C01819=1049.638,44.373,421.280,170.592,33.562,156.310
C01820=1049.643,44.623,421.263,170.594,33.564,156.311
C01821=1049.650,44.872,421.246,170.596,33.566,156.311
C01822=1049.656,45.158,421.226,170.597,33.568,156.311
C01823=1049.664,45.444,421.207,170.599,33.571,156.312
C01824=1049.671,45.731,421.188,170.601,33.573,156.312
C01825=1049.678,46.017,421.168,170.603,33.575,156.312
C01826=1049.684,46.266,421.152,170.605,33.577,156.313
C01827=1049.690,46.516,421.134,170.606,33.579,156.313
C01828=1049.696,46.765,421.117,170.608,33.581,156.313
C01829=1049.702,47.014,421.100,170.610,33.583,156.314
C01830=1049.709,47.263,421.083,170.611,33.585,156.314
C01831=1049.714,47.513,421.066,170.613,33.587,156.314
C01832=1049.721,47.762,421.049,170.615,33.589,156.315
C01833=1049.727,48.012,421.033,170.617,33.590,156.315
C01834=1049.732,48.261,421.015,170.619,33.592,156.315
C01835=1049.739,48.510,420.998,170.620,33.594,156.316
C01836=1049.745,48.759,420.982,170.622,33.596,156.316
C01837=1049.751,49.008,420.964,170.624,33.598,156.316
C01838=1049.757,49.258,420.947,170.625,33.600,156.316
C01839=1049.763,49.507,420.930,170.627,33.602,156.317
C01840=1049.770,49.757,420.912,170.629,33.604,156.317
C01841=1049.775,50.006,420.896,170.630,33.606,156.317
C01842=1049.781,50.255,420.879,170.632,33.608,156.318
C01843=1049.788,50.505,420.861,170.634,33.610,156.318
C01844=1049.794,50.754,420.845,170.635,33.612,156.318
C01845=1049.800,51.004,420.827,170.637,33.614,156.319
C01846=1049.806,51.253,420.810,170.638,33.616,156.319
C01847=1049.813,51.503,420.793,170.640,33.618,156.319
C01848=1049.818,51.752,420.776,170.642,33.620,156.320
C01849=1049.825,52.001,420.759,170.643,33.622,156.320
C01850=1049.831,52.250,420.742,170.645,33.624,156.320
C01851=1049.837,52.499,420.725,170.647,33.626,156.321
C01852=1049.843,52.749,420.707,170.648,33.628,156.321
C01853=1049.850,52.998,420.690,170.650,33.630,156.321
C01854=1049.856,53.247,420.673,170.652,33.632,156.322
C01855=1049.862,53.497,420.656,170.653,33.633,156.322
C01856=1049.868,53.746,420.638,170.655,33.635,156.322
C01857=1049.874,53.995,420.621,170.656,33.637,156.322
C01858=1049.881,54.245,420.604,170.658,33.639,156.323
C01859=1049.886,54.494,420.587,170.660,33.641,156.323
C01860=1049.893,54.744,420.570,170.661,33.643,156.323
C01861=1049.899,54.992,420.553,170.663,33.645,156.324
C01862=1049.905,55.242,420.535,170.665,33.647,156.324
C01863=1049.912,55.491,420.518,170.666,33.649,156.324
C01864=1049.918,55.741,420.501,170.668,33.651,156.325
C01865=1049.924,55.990,420.484,170.670,33.653,156.325
C01866=1049.931,56.239,420.466,170.671,33.655,156.325
C01867=1049.936,56.488,420.449,170.673,33.657,156.326
C01868=1049.943,56.738,420.432,170.674,33.659,156.326
C01869=1049.949,56.988,420.414,170.676,33.660,156.326
C01870=1049.955,57.236,420.397,170.678,33.662,156.326
C01871=1049.962,57.486,420.380,170.679,33.664,156.327
C01872=1049.967,57.735,420.362,170.681,33.666,156.327
C01873=1049.974,57.985,420.345,170.684,33.668,156.327
C01874=1049.980,58.234,420.328,170.685,33.670,156.328
C01875=1049.987,58.483,420.310,170.687,33.672,156.328
C01876=1049.994,58.733,420.293,170.689,33.674,156.328
C01877=1049.999,58.982,420.275,170.690,33.676,156.329
C01878=1050.006,59.231,420.258,170.692,33.678,156.329
C01879=1050.011,59.480,420.240,170.693,33.680,156.329
C01880=1050.018,59.730,420.223,170.695,33.682,156.330
C01881=1050.024,59.979,420.205,170.697,33.683,156.330
C01882=1050.031,60.228,420.188,170.698,33.685,156.330
C01883=1050.038,60.478,420.171,170.700,33.687,156.330
C01884=1050.043,60.727,420.153,170.702,33.689,156.331
C01885=1050.050,60.976,420.136,170.703,33.691,156.331
C01886=1050.057,61.262,420.116,170.705,33.693,156.331
C01887=1050.064,61.548,420.096,170.707,33.696,156.332
C01888=1050.071,61.834,420.076,170.709,33.698,156.332
C01889=1050.079,62.120,420.057,170.711,33.700,156.332
C01890=1050.085,62.369,420.039,170.712,33.702,156.333
C01891=1050.091,62.619,420.021,170.714,33.704,156.333
C01892=1050.097,62.868,420.004,170.716,33.706,156.333
C01893=1050.104,63.117,419.986,170.717,33.708,156.334
C01894=1050.110,63.366,419.968,170.719,33.710,156.334
C01895=1050.117,63.615,419.951,170.721,33.712,156.334
C01896=1050.123,63.865,419.933,170.722,33.713,156.335
C01897=1050.130,64.114,419.916,170.724,33.715,156.335
C01898=1050.135,64.363,419.898,170.726,33.717,156.335
C01899=1050.142,64.613,419.881,170.727,33.719,156.336
C01900=1050.148,64.862,419.863,170.729,33.721,156.336
C01901=1050.154,65.111,419.845,170.730,33.723,156.336
C01902=1050.160,65.361,419.827,170.732,33.725,156.337
C01903=1050.167,65.610,419.809,170.734,33.727,156.337
C01904=1050.172,65.859,419.792,170.735,33.729,156.337
C01905=1050.178,66.109,419.774,170.737,33.731,156.337
C01906=1050.185,66.358,419.756,170.739,33.733,156.338
C01907=1050.191,66.607,419.739,170.741,33.734,156.338
C01908=1050.197,66.856,419.720,170.743,33.736,156.338
C01909=1050.204,67.106,419.703,170.744,33.738,156.339
C01910=1050.210,67.355,419.685,170.746,33.741,156.339
C01911=1050.216,67.605,419.667,170.748,33.743,156.340
C01912=1050.222,67.854,419.649,170.749,33.745,156.340
C01913=1050.228,68.102,419.632,170.751,33.747,156.340
C01914=1050.235,68.352,419.614,170.753,33.749,156.340
C01915=1050.241,68.602,419.596,170.754,33.751,156.341
C01916=1050.247,68.850,419.578,170.756,33.753,156.341
C01917=1050.253,69.100,419.560,170.757,33.755,156.341
C01918=1050.259,69.350,419.542,170.759,33.757,156.342
C01919=1050.265,69.599,419.525,170.761,33.759,156.342
C01920=1050.271,69.848,419.506,170.762,33.761,156.342
C01921=1050.278,70.097,419.488,170.764,33.763,156.343
C01922=1050.283,70.346,419.471,170.766,33.764,156.343
C01923=1050.290,70.596,419.452,170.767,33.766,156.343
C01924=1050.296,70.845,419.435,170.769,33.768,156.344
C01925=1050.302,71.094,419.417,170.770,33.770,156.344
C01926=1050.308,71.343,419.398,170.772,33.772,156.344
C01927=1050.314,71.593,419.380,170.774,33.774,156.345
C01928=1050.321,71.843,419.362,170.775,33.776,156.345
C01929=1050.326,72.091,419.344,170.777,33.778,156.345
C01930=1050.332,72.341,419.326,170.779,33.780,156.346
C01931=1050.339,72.590,419.308,170.780,33.783,156.346
C01932=1050.345,72.840,419.290,170.782,33.785,156.346
C01933=1050.351,73.088,419.273,170.783,33.787,156.347
C01934=1050.358,73.338,419.254,170.786,33.789,156.347
C01935=1050.364,73.587,419.236,170.788,33.791,156.347
C01936=1050.370,73.836,419.218,170.789,33.792,156.348
C01937=1050.376,74.085,419.200,170.791,33.794,156.348
C01938=1050.382,74.335,419.181,170.792,33.796,156.348
C01939=1050.388,74.584,419.163,170.794,33.798,156.349
C01940=1050.395,74.833,419.145,170.796,33.800,156.349
C01941=1050.400,75.082,419.127,170.797,33.802,156.349
C01942=1050.407,75.332,419.108,170.799,33.804,156.350
C01943=1050.413,75.581,419.091,170.801,33.806,156.350
C01944=1050.419,75.830,419.072,170.802,33.808,156.350
C01945=1050.425,76.079,419.054,170.804,33.810,156.351
C01946=1050.431,76.329,419.036,170.805,33.812,156.351
C01947=1050.437,76.578,419.018,170.807,33.814,156.351
C01948=1050.444,76.827,419.000,170.809,33.816,156.352
C01949=1050.451,77.077,418.982,170.810,33.819,156.352
C01950=1050.457,77.363,418.960,170.812,33.821,156.352
C01951=1050.464,77.648,418.940,170.814,33.823,156.353
C01952=1050.471,77.933,418.919,170.816,33.825,156.353
C01953=1050.479,78.219,418.898,170.818,33.828,156.353
C01954=1050.484,78.468,418.880,170.819,33.830,156.354
C01955=1050.491,78.718,418.861,170.821,33.832,156.354
C01956=1050.496,78.967,418.842,170.823,33.834,156.354
C01957=1050.503,79.217,418.824,170.824,33.835,156.355
C01958=1050.509,79.466,418.805,170.827,33.837,156.355
C01959=1050.515,79.714,418.787,170.828,33.839,156.355
C01960=1050.521,79.964,418.769,170.830,33.842,156.356
C01961=1050.527,80.213,418.751,170.832,33.844,156.356
C01962=1050.533,80.463,418.731,170.833,33.846,156.357
C01963=1050.539,80.712,418.713,170.835,33.848,156.357
C01964=1050.545,80.961,418.695,170.837,33.850,156.357
C01965=1050.551,81.210,418.677,170.838,33.852,156.357
C01966=1050.558,81.460,418.659,170.840,33.854,156.358
C01967=1050.563,81.709,418.639,170.841,33.856,156.358
C01968=1050.570,81.958,418.621,170.843,33.858,156.359
C01969=1050.576,82.207,418.602,170.845,33.860,156.359
C01970=1050.582,82.456,418.584,170.846,33.862,156.359
C01971=1050.588,82.705,418.566,170.848,33.864,156.360
C01972=1050.594,82.955,418.547,170.849,33.866,156.360
C01973=1050.600,83.204,418.528,170.851,33.868,156.360
C01974=1050.606,83.454,418.510,170.853,33.871,156.361
C01975=1050.613,83.703,418.491,170.854,33.872,156.361
C01976=1050.618,83.952,418.472,170.856,33.874,156.361
C01977=1050.624,84.201,418.454,170.858,33.876,156.362
C01978=1050.630,84.450,418.436,170.859,33.878,156.362
C01979=1050.637,84.700,418.417,170.861,33.880,156.362
C01980=1050.643,84.949,418.399,170.863,33.882,156.363
C01981=1050.649,85.198,418.379,170.865,33.884,156.363
C01982=1050.655,85.447,418.361,170.867,33.887,156.363
C01983=1050.662,85.696,418.342,170.868,33.889,156.364
C01984=1050.668,85.946,418.324,170.870,33.891,156.364
C01985=1050.674,86.196,418.305,170.872,33.893,156.364
C01986=1050.680,86.445,418.286,170.873,33.895,156.365
C01987=1050.686,86.693,418.268,170.875,33.896,156.365
C01988=1050.692,86.942,418.249,170.876,33.898,156.365
C01989=1050.699,87.191,418.231,170.878,33.900,156.366
C01990=1050.704,87.441,418.211,170.880,33.902,156.366
C01991=1050.711,87.690,418.193,170.881,33.905,156.366
C01992=1050.717,87.940,418.175,170.883,33.907,156.367
C01993=1050.723,88.189,418.156,170.885,33.909,156.367
C01994=1050.729,88.438,418.137,170.886,33.911,156.367
C01995=1050.735,88.687,418.118,170.888,33.913,156.368
C01996=1050.742,88.936,418.100,170.890,33.915,156.368
C01997=1050.748,89.186,418.081,170.891,33.917,156.368
C01998=1050.754,89.435,418.062,170.893,33.919,156.369
C01999=1050.760,89.684,418.043,170.894,33.920,156.369
C02000=1050.767,89.933,418.024,170.896,33.922,156.369
C02001=1050.772,90.183,418.005,170.898,33.924,156.370
C02002=1050.779,90.432,417.987,170.900,33.926,156.370
C02003=1050.785,90.681,417.968,170.902,33.929,156.370
C02004=1050.791,90.930,417.949,170.904,33.931,156.371
C02005=1050.797,91.179,417.930,170.905,33.933,156.371
C02006=1050.803,91.429,417.911,170.907,33.935,156.371
C02007=1050.810,91.678,417.892,170.908,33.937,156.372
C02008=1050.815,91.927,417.873,170.910,33.939,156.372
C02009=1050.822,92.177,417.854,170.912,33.941,156.372
C02010=1050.827,92.426,417.835,170.913,33.943,156.373
C02011=1050.834,92.675,417.816,170.915,33.945,156.373
C02012=1050.840,92.924,417.796,170.917,33.948,156.374
C02013=1050.846,93.173,417.778,170.918,33.950,156.374
C02014=1050.853,93.459,417.756,170.920,33.952,156.374
C02015=1050.860,93.744,417.734,170.922,33.954,156.375
C02016=1050.867,94.030,417.713,170.924,33.957,156.375
C02017=1050.874,94.315,417.691,170.926,33.959,156.375
C02018=1050.879,94.564,417.672,170.927,33.961,156.376
C02019=1050.886,94.814,417.653,170.929,33.963,156.376
C02020=1050.891,95.063,417.634,170.932,33.965,156.376
C02021=1050.897,95.312,417.614,170.933,33.967,156.377
C02022=1050.904,95.562,417.595,170.935,33.969,156.377
C02023=1050.910,95.811,417.576,170.937,33.972,156.378
C02024=1050.916,96.060,417.557,170.938,33.973,156.378
C02025=1050.922,96.310,417.538,170.940,33.975,156.378
C02026=1050.929,96.558,417.518,170.941,33.977,156.379
C02027=1050.935,96.808,417.499,170.943,33.979,156.379
C02028=1050.941,97.057,417.480,170.945,33.981,156.379
C02029=1050.947,97.306,417.461,170.946,33.984,156.380
C02030=1050.953,97.555,417.442,170.948,33.986,156.380
C02031=1050.959,97.804,417.423,170.950,33.988,156.380
C02032=1050.965,98.053,417.403,170.951,33.990,156.381
C02033=1050.971,98.303,417.385,170.953,33.992,156.381
C02034=1050.977,98.552,417.365,170.955,33.994,156.381
C02035=1050.984,98.801,417.346,170.956,33.996,156.382
C02036=1050.989,99.050,417.327,170.958,33.998,156.382
C02037=1050.996,99.300,417.308,170.960,34.000,156.382
C02038=1051.002,99.549,417.288,170.962,34.002,156.383
C02039=1051.009,99.798,417.269,170.964,34.004,156.383
C02040=1051.014,100.047,417.250,170.966,34.006,156.383
C02041=1051.020,100.296,417.230,170.967,34.008,156.384
C02042=1051.027,100.545,417.211,170.969,34.010,156.384
C02043=1051.033,100.795,417.192,170.970,34.012,156.384
C02044=1051.039,101.043,417.172,170.972,34.014,156.385
C02045=1051.045,101.292,417.153,170.974,34.016,156.385
C02046=1051.051,101.542,417.134,170.975,34.019,156.386
C02047=1051.057,101.791,417.114,170.977,34.021,156.386
C02048=1051.063,102.041,417.095,170.979,34.023,156.386
C02049=1051.069,102.290,417.075,170.980,34.024,156.387
C02050=1051.075,102.539,417.056,170.982,34.027,156.387
C02051=1051.081,102.788,417.036,170.984,34.029,156.387
C02052=1051.087,103.037,417.017,170.985,34.031,156.388
C02053=1051.093,103.286,416.997,170.987,34.033,156.388
C02054=1051.099,103.535,416.978,170.989,34.035,156.388
C02055=1051.105,103.784,416.958,170.991,34.037,156.389
C02056=1051.111,104.033,416.939,170.993,34.039,156.389
C02057=1051.117,104.283,416.919,170.995,34.042,156.389
C02058=1051.123,104.532,416.899,170.996,34.044,156.390
C02059=1051.129,104.782,416.880,170.998,34.046,156.390
C02060=1051.135,105.030,416.860,170.999,34.048,156.390
C02061=1051.142,105.279,416.841,171.001,34.050,156.391
C02062=1051.148,105.528,416.822,171.003,34.052,156.391
C02063=1051.154,105.777,416.802,171.004,34.054,156.392
C02064=1051.160,106.027,416.782,171.006,34.056,156.392
C02065=1051.166,106.276,416.762,171.008,34.059,156.392
C02066=1051.172,106.526,416.743,171.009,34.060,156.393
C02067=1051.178,106.774,416.724,171.011,34.062,156.393
C02068=1051.184,107.023,416.704,171.013,34.064,156.393
C02069=1051.191,107.273,416.684,171.014,34.066,156.394
C02070=1051.197,107.522,416.664,171.016,34.069,156.394
C02071=1051.202,107.771,416.645,171.019,34.071,156.394
C02072=1051.208,108.020,416.625,171.020,34.073,156.395
C02073=1051.215,108.269,416.606,171.022,34.075,156.395
C02074=1051.221,108.519,416.586,171.024,34.077,156.396
C02075=1051.227,108.767,416.566,171.025,34.079,156.396
C02076=1051.233,109.017,416.547,171.027,34.081,156.396
C02077=1051.239,109.266,416.527,171.029,34.083,156.397
C02078=1051.246,109.551,416.504,171.031,34.086,156.397
C02079=1051.253,109.837,416.481,171.033,34.088,156.397
C02080=1051.260,110.123,416.459,171.035,34.090,156.398
C02081=1051.267,110.408,416.436,171.036,34.093,156.398
C02082=1051.274,110.658,416.417,171.038,34.095,156.399
C02083=1051.280,110.906,416.397,171.040,34.097,156.399
C02084=1051.286,111.155,416.377,171.041,34.099,156.399
C02085=1051.292,111.405,416.358,171.043,34.101,156.400
C02086=1051.298,111.654,416.337,171.045,34.103,156.400
C02087=1051.304,111.903,416.317,171.048,34.105,156.400
C02088=1051.310,112.152,416.297,171.049,34.107,156.401
C02089=1051.316,112.401,416.278,171.051,34.109,156.401
C02090=1051.322,112.651,416.258,171.053,34.111,156.401
C02091=1051.328,112.900,416.238,171.054,34.114,156.402
C02092=1051.334,113.148,416.218,171.056,34.116,156.402
C02093=1051.340,113.397,416.198,171.058,34.118,156.402
C02094=1051.347,113.647,416.178,171.059,34.120,156.403
C02095=1051.353,113.896,416.158,171.061,34.122,156.403
C02096=1051.358,114.145,416.138,171.063,34.124,156.404
C02097=1051.364,114.394,416.118,171.064,34.126,156.404
C02098=1051.371,114.644,416.097,171.066,34.129,156.404
C02099=1051.377,114.892,416.078,171.068,34.131,156.405
C02100=1051.382,115.142,416.057,171.069,34.133,156.405
C02101=1051.388,115.390,416.037,171.072,34.135,156.405
C02102=1051.394,115.641,416.017,171.074,34.137,156.406
C02103=1051.399,115.890,415.997,171.075,34.139,156.406
C02104=1051.405,116.138,415.977,171.077,34.141,156.407
C02105=1051.411,116.387,415.957,171.079,34.144,156.407
C02106=1051.418,116.637,415.937,171.080,34.146,156.407
C02107=1051.423,116.886,415.916,171.082,34.148,156.408
C02108=1051.429,117.135,415.896,171.084,34.150,156.408
C02109=1051.436,117.384,415.876,171.085,34.152,156.408
C02110=1051.442,117.633,415.856,171.087,34.154,156.409
C02111=1051.447,117.882,415.835,171.089,34.157,156.409
C02112=1051.453,118.131,415.815,171.090,34.159,156.410
C02113=1051.460,118.381,415.795,171.092,34.161,156.410
C02114=1051.466,118.629,415.775,171.094,34.163,156.410
C02115=1051.471,118.878,415.754,171.096,34.165,156.411
C02116=1051.477,119.128,415.734,171.098,34.168,156.411
C02117=1051.483,119.377,415.714,171.100,34.170,156.411
C02118=1051.489,119.626,415.694,171.102,34.172,156.412
C02119=1051.495,119.875,415.673,171.103,34.174,156.412
C02120=1051.501,120.124,415.653,171.105,34.176,156.413
C02121=1051.507,120.373,415.633,171.107,34.179,156.413
C02122=1051.513,120.623,415.612,171.108,34.180,156.413
C02123=1051.519,120.871,415.592,171.110,34.182,156.414
C02124=1051.525,121.120,415.572,171.112,34.185,156.414
C02125=1051.531,121.370,415.551,171.113,34.187,156.414
C02126=1051.537,121.619,415.531,171.115,34.189,156.415
C02127=1051.543,121.867,415.511,171.117,34.191,156.415
C02128=1051.549,122.117,415.490,171.119,34.193,156.416
C02129=1051.555,122.366,415.470,171.121,34.195,156.416
C02130=1051.562,122.615,415.450,171.123,34.198,156.416
C02131=1051.567,122.864,415.429,171.125,34.200,156.417
C02132=1051.573,123.113,415.409,171.126,34.202,156.417
C02133=1051.580,123.362,415.388,171.128,34.204,156.417
C02134=1051.585,123.611,415.368,171.130,34.206,156.418
C02135=1051.592,123.861,415.347,171.132,34.208,156.418
C02136=1051.598,124.110,415.327,171.133,34.211,156.419
C02137=1051.604,124.358,415.307,171.135,34.212,156.419
C02138=1051.610,124.608,415.286,171.137,34.214,156.419
C02139=1051.616,124.857,415.266,171.138,34.217,156.420
C02140=1051.622,125.106,415.246,171.140,34.219,156.420
C02141=1051.628,125.355,415.225,171.142,34.221,156.420
C02142=1051.635,125.641,415.201,171.145,34.223,156.421
C02143=1051.642,125.926,415.178,171.147,34.226,156.421
C02144=1051.649,126.211,415.154,171.149,34.228,156.422
C02145=1051.656,126.497,415.130,171.151,34.231,156.422
C02146=1051.662,126.746,415.110,171.153,34.233,156.422
C02147=1051.668,126.995,415.090,171.154,34.235,156.423
C02148=1051.675,127.244,415.068,171.156,34.237,156.423
C02149=1051.681,127.493,415.048,171.158,34.239,156.423
C02150=1051.687,127.743,415.028,171.160,34.241,156.424
C02151=1051.693,127.991,415.007,171.161,34.243,156.424
C02152=1051.699,128.241,414.987,171.163,34.246,156.425
C02153=1051.705,128.490,414.966,171.165,34.248,156.425
C02154=1051.711,128.739,414.945,171.167,34.250,156.425
C02155=1051.717,128.988,414.925,171.169,34.252,156.426
C02156=1051.723,129.237,414.904,171.171,34.254,156.426
C02157=1051.730,129.486,414.883,171.173,34.256,156.426
C02158=1051.736,129.735,414.863,171.175,34.259,156.427
C02159=1051.741,129.984,414.843,171.176,34.260,156.427
C02160=1051.748,130.233,414.821,171.178,34.262,156.427
C02161=1051.754,130.482,414.802,171.180,34.265,156.428
C02162=1051.760,130.731,414.780,171.182,34.267,156.428
C02163=1051.766,130.980,414.760,171.183,34.269,156.429
C02164=1051.772,131.230,414.739,171.185,34.271,156.429
C02165=1051.779,131.479,414.718,171.187,34.273,156.429
C02166=1051.784,131.728,414.697,171.189,34.275,156.430
C02167=1051.791,131.977,414.676,171.191,34.278,156.430
C02168=1051.797,132.226,414.656,171.193,34.280,156.430
C02169=1051.803,132.475,414.634,171.195,34.282,156.431
C02170=1051.809,132.724,414.614,171.197,34.284,156.431
C02171=1051.815,132.973,414.593,171.198,34.286,156.432
C02172=1051.820,133.222,414.572,171.200,34.289,156.432
C02173=1051.827,133.471,414.551,171.202,34.290,156.432
C02174=1051.833,133.720,414.530,171.204,34.293,156.433
C02175=1051.839,133.969,414.509,171.205,34.295,156.433
C02176=1051.845,134.218,414.488,171.207,34.297,156.434
C02177=1051.851,134.467,414.467,171.209,34.299,156.434
C02178=1051.857,134.717,414.446,171.211,34.301,156.434
C02179=1051.863,134.965,414.426,171.213,34.304,156.435
C02180=1051.869,135.215,414.404,171.215,34.306,156.435
C02181=1051.875,135.463,414.383,171.217,34.308,156.436
C02182=1051.881,135.713,414.362,171.219,34.310,156.436
C02183=1051.887,135.961,414.341,171.221,34.313,156.436
C02184=1051.893,136.210,414.319,171.222,34.315,156.437
C02185=1051.900,136.460,414.299,171.224,34.317,156.437
C02186=1051.905,136.708,414.278,171.226,34.319,156.437
C02187=1051.911,136.958,414.256,171.228,34.321,156.438
C02188=1051.917,137.206,414.236,171.229,34.324,156.438
C02189=1051.923,137.456,414.215,171.231,34.325,156.439
C02190=1051.930,137.705,414.193,171.233,34.328,156.439
C02191=1051.935,137.954,414.172,171.236,34.330,156.439
C02192=1051.942,138.203,414.151,171.238,34.332,156.440
C02193=1051.947,138.451,414.130,171.239,34.334,156.440
C02194=1051.953,138.700,414.109,171.241,34.336,156.440
C02195=1051.959,138.950,414.088,171.243,34.339,156.441
C02196=1051.966,139.199,414.067,171.245,34.341,156.441
C02197=1051.972,139.448,414.045,171.246,34.343,156.442
C02198=1051.978,139.697,414.024,171.248,34.345,156.442
C02199=1051.983,139.946,414.003,171.250,34.348,156.442
C02200=1051.989,140.195,413.981,171.252,34.350,156.443
C02201=1051.995,140.444,413.960,171.254,34.352,156.443
C02202=1052.001,140.693,413.939,171.256,34.354,156.444
C02203=1052.008,140.942,413.918,171.258,34.357,156.444
C02204=1052.013,141.191,413.897,171.260,34.359,156.444
C02205=1052.019,141.440,413.875,171.262,34.361,156.445
C02206=1052.026,141.725,413.850,171.264,34.364,156.445
C02207=1052.033,142.010,413.826,171.266,34.366,156.446
C02208=1052.040,142.296,413.802,171.268,34.369,156.446
C02209=1052.047,142.582,413.776,171.270,34.371,156.447
C02210=1052.052,142.830,413.755,171.272,34.373,156.447
C02211=1052.059,143.079,413.734,171.274,34.376,156.447
C02212=1052.065,143.329,413.713,171.276,34.378,156.448
C02213=1052.071,143.577,413.692,171.278,34.380,156.448
C02214=1052.077,143.826,413.670,171.280,34.382,156.448
C02215=1052.083,144.076,413.649,171.282,34.385,156.449
C02216=1052.088,144.324,413.627,171.284,34.387,156.449
C02217=1052.095,144.573,413.606,171.285,34.389,156.450
C02218=1052.101,144.823,413.584,171.287,34.392,156.450
C02219=1052.106,145.071,413.563,171.289,34.393,156.450
C02220=1052.113,145.320,413.541,171.291,34.396,156.451
C02221=1052.119,145.569,413.520,171.293,34.398,156.451
C02222=1052.125,145.819,413.498,171.295,34.400,156.452
C02223=1052.130,146.067,413.477,171.297,34.402,156.452
C02224=1052.137,146.316,413.455,171.299,34.405,156.453
C02225=1052.143,146.566,413.433,171.301,34.407,156.453
C02226=1052.149,146.815,413.412,171.303,34.409,156.453
C02227=1052.154,147.063,413.390,171.305,34.411,156.454
C02228=1052.161,147.313,413.369,171.307,34.414,156.454
C02229=1052.167,147.562,413.347,171.308,34.416,156.454
C02230=1052.173,147.810,413.325,171.310,34.418,156.455
C02231=1052.179,148.059,413.304,171.312,34.420,156.455
C02232=1052.185,148.308,413.282,171.314,34.423,156.456
C02233=1052.191,148.557,413.260,171.317,34.425,156.456
C02234=1052.197,148.806,413.239,171.319,34.427,156.456
C02235=1052.203,149.055,413.217,171.320,34.430,156.457
C02236=1052.209,149.304,413.196,171.322,34.432,156.457
C02237=1052.215,149.553,413.173,171.324,34.434,156.458
C02238=1052.221,149.802,413.151,171.326,34.436,156.458
C02239=1052.226,150.051,413.130,171.328,34.439,156.458
C02240=1052.233,150.300,413.108,171.330,34.440,156.459
C02241=1052.239,150.549,413.087,171.332,34.443,156.459
C02242=1052.245,150.798,413.064,171.333,34.445,156.460
C02243=1052.251,151.047,413.042,171.336,34.447,156.460
C02244=1052.256,151.296,413.021,171.338,34.450,156.460
C02245=1052.262,151.545,412.999,171.340,34.452,156.461
C02246=1052.269,151.794,412.978,171.342,34.454,156.461
C02247=1052.275,152.043,412.955,171.344,34.457,156.462
C02248=1052.280,152.292,412.933,171.345,34.459,156.462
C02249=1052.286,152.541,412.912,171.347,34.461,156.463
C02250=1052.293,152.789,412.889,171.349,34.463,156.463
C02251=1052.299,153.039,412.868,171.351,34.466,156.463
C02252=1052.305,153.288,412.846,171.353,34.468,156.464
C02253=1052.311,153.537,412.823,171.356,34.470,156.464
C02254=1052.317,153.786,412.801,171.358,34.473,156.465
C02255=1052.322,154.034,412.780,171.360,34.475,156.465
C02256=1052.329,154.283,412.758,171.361,34.477,156.465
C02257=1052.335,154.532,412.736,171.363,34.480,156.466
C02258=1052.340,154.782,412.714,171.365,34.482,156.466
C02259=1052.347,155.030,412.692,171.367,34.484,156.467
C02260=1052.353,155.279,412.670,171.369,34.487,156.467
C02261=1052.358,155.529,412.648,171.371,34.489,156.467
C02262=1052.364,155.777,412.626,171.373,34.491,156.468
C02263=1052.370,156.026,412.604,171.376,34.494,156.468
C02264=1052.376,156.275,412.581,171.377,34.495,156.469
C02265=1052.382,156.524,412.560,171.379,34.498,156.469
C02266=1052.389,156.773,412.537,171.381,34.501,156.470
C02267=1052.394,157.022,412.515,171.383,34.502,156.470
C02268=1052.401,157.271,412.493,171.385,34.505,156.470
C02269=1052.406,157.520,412.470,171.387,34.507,156.471
C02270=1052.413,157.805,412.445,171.389,34.510,156.471
C02271=1052.420,158.090,412.420,171.391,34.513,156.472
C02272=1052.426,158.375,412.395,171.394,34.515,156.472
C02273=1052.434,158.660,412.369,171.397,34.518,156.473
C02274=1052.440,158.909,412.347,171.399,34.520,156.473
C02275=1052.446,159.158,412.325,171.400,34.523,156.473
C02276=1052.451,159.407,412.303,171.402,34.525,156.474
C02277=1052.458,159.655,412.281,171.404,34.527,156.474
C02278=1052.463,159.904,412.258,171.406,34.530,156.475
C02279=1052.469,160.153,412.236,171.408,34.531,156.475
C02280=1052.476,160.402,412.214,171.411,34.534,156.475
C02281=1052.481,160.652,412.191,171.413,34.537,156.476
C02282=1052.488,160.900,412.169,171.415,34.538,156.476
C02283=1052.494,161.149,412.146,171.417,34.541,156.477
C02284=1052.499,161.399,412.124,171.419,34.543,156.477
C02285=1052.505,161.647,412.101,171.421,34.546,156.478
C02286=1052.511,161.896,412.079,171.422,34.548,156.478
C02287=1052.517,162.146,412.056,171.424,34.551,156.479
C02288=1052.522,162.394,412.033,171.426,34.554,156.479
C02289=1052.527,162.643,412.011,171.429,34.555,156.479
C02290=1052.534,162.891,411.988,171.431,34.558,156.480
C02291=1052.539,163.141,411.966,171.433,34.560,156.480
C02292=1052.545,163.390,411.943,171.435,34.563,156.481
C02293=1052.551,163.639,411.920,171.437,34.565,156.481
C02294=1052.557,163.887,411.898,171.439,34.568,156.482
C02295=1052.563,164.137,411.876,171.441,34.571,156.482
C02296=1052.568,164.386,411.853,171.442,34.573,156.483
C02297=1052.574,164.634,411.830,171.445,34.575,156.483
C02298=1052.581,164.883,411.808,171.447,34.577,156.483
C02299=1052.586,165.132,411.785,171.449,34.580,156.484
C02300=1052.592,165.381,411.762,171.451,34.582,156.484
C02301=1052.598,165.630,411.739,171.453,34.585,156.485
C02302=1052.603,165.879,411.716,171.455,34.587,156.485
C02303=1052.610,166.128,411.694,171.457,34.590,156.486
C02304=1052.615,166.377,411.671,171.459,34.592,156.486
C02305=1052.621,166.626,411.648,171.461,34.594,156.486
C02306=1052.627,166.875,411.625,171.464,34.597,156.487
C02307=1052.633,167.123,411.603,171.466,34.599,156.487
C02308=1052.639,167.372,411.580,171.468,34.602,156.488
C02309=1052.645,167.622,411.558,171.470,34.604,156.488
C02310=1052.650,167.870,411.535,171.472,34.607,156.489
C02311=1052.656,168.119,411.512,171.474,34.610,156.489
C02312=1052.662,168.368,411.489,171.476,34.611,156.489
C02313=1052.668,168.617,411.467,171.477,34.614,156.490
C02314=1052.674,168.866,411.444,171.480,34.616,156.490
C02315=1052.680,169.115,411.421,171.482,34.619,156.491
C02316=1052.685,169.364,411.398,171.484,34.621,156.491
C02317=1052.691,169.612,411.375,171.486,34.624,156.492
C02318=1052.698,169.861,411.352,171.488,34.626,156.492
C02319=1052.703,170.110,411.329,171.490,34.628,156.493
C02320=1052.709,170.359,411.307,171.492,34.631,156.493
C02321=1052.715,170.608,411.284,171.494,34.633,156.493
C02322=1052.721,170.857,411.261,171.497,34.636,156.494
C02323=1052.727,171.105,411.238,171.499,34.638,156.494
C02324=1052.733,171.355,411.215,171.501,34.641,156.495
C02325=1052.739,171.603,411.191,171.503,34.643,156.495
C02326=1052.745,171.852,411.168,171.505,34.646,156.496
C02327=1052.751,172.101,411.145,171.507,34.648,156.496
C02328=1052.757,172.350,411.122,171.509,34.650,156.497
C02329=1052.763,172.598,411.100,171.511,34.653,156.497
C02330=1052.769,172.847,411.077,171.514,34.655,156.497
C02331=1052.774,173.096,411.054,171.516,34.658,156.498
C02332=1052.781,173.346,411.031,171.518,34.660,156.498
C02333=1052.787,173.595,411.008,171.520,34.663,156.499
C02334=1052.794,173.878,410.982,171.523,34.665,156.499
C02335=1052.800,174.163,410.955,171.525,34.669,156.500
C02336=1052.808,174.448,410.929,171.527,34.671,156.500
C02337=1052.814,174.732,410.902,171.530,34.674,156.501
C02338=1052.820,174.981,410.879,171.532,34.676,156.501
C02339=1052.826,175.230,410.857,171.534,34.679,156.502
C02340=1052.832,175.478,410.833,171.537,34.681,156.502
C02341=1052.838,175.728,410.810,171.539,34.684,156.503
C02342=1052.844,175.977,410.787,171.541,34.686,156.503
C02343=1052.850,176.226,410.764,171.543,34.689,156.504
C02344=1052.856,176.474,410.740,171.546,34.691,156.504
C02345=1052.862,176.724,410.717,171.548,34.694,156.504
C02346=1052.868,176.972,410.694,171.550,34.696,156.505
C02347=1052.875,177.220,410.671,171.552,34.698,156.505
C02348=1052.880,177.469,410.648,171.554,34.701,156.506
C02349=1052.887,177.719,410.625,171.556,34.703,156.506
C02350=1052.893,177.967,410.601,171.558,34.706,156.507
C02351=1052.899,178.216,410.578,171.560,34.708,156.507
C02352=1052.904,178.465,410.555,171.563,34.711,156.508
C02353=1052.911,178.714,410.531,171.565,34.713,156.508
C02354=1052.917,178.963,410.508,171.567,34.716,156.508
C02355=1052.922,179.212,410.485,171.569,34.717,156.509
C02356=1052.929,179.461,410.461,171.571,34.720,156.509
C02357=1052.936,179.709,410.439,171.573,34.722,156.510
C02358=1052.941,179.958,410.416,171.575,34.725,156.510
C02359=1052.947,180.206,410.392,171.578,34.727,156.511
C02360=1052.954,180.456,410.369,171.581,34.730,156.511
C02361=1052.960,180.704,410.345,171.583,34.732,156.512
C02362=1052.965,180.953,410.322,171.585,34.735,156.512
C02363=1052.972,181.202,410.298,171.587,34.737,156.512
C02364=1052.978,181.451,410.275,171.589,34.740,156.513
C02365=1052.984,181.699,410.252,171.591,34.742,156.513
C02366=1052.990,181.949,410.229,171.593,34.744,156.514
C02367=1052.996,182.197,410.205,171.596,34.747,156.514
C02368=1053.002,182.447,410.182,171.598,34.749,156.515
C02369=1053.009,182.695,410.158,171.600,34.752,156.515
C02370=1053.015,182.944,410.136,171.603,34.754,156.516
C02371=1053.022,183.193,410.112,171.605,34.757,156.516
C02372=1053.027,183.442,410.089,171.607,34.759,156.516
C02373=1053.033,183.690,410.065,171.609,34.762,156.517
C02374=1053.040,183.939,410.042,171.612,34.764,156.517
C02375=1053.046,184.188,410.018,171.614,34.767,156.518
C02376=1053.051,184.438,409.994,171.616,34.769,156.518
C02377=1053.057,184.686,409.970,171.618,34.772,156.519
C02378=1053.063,184.935,409.946,171.620,34.774,156.519
C02379=1053.068,185.183,409.923,171.622,34.777,156.520
C02380=1053.075,185.432,409.899,171.625,34.780,156.520
C02381=1053.080,185.681,409.875,171.628,34.783,156.521
C02382=1053.086,185.929,409.851,171.630,34.785,156.521
C02383=1053.092,186.179,409.827,171.632,34.788,156.522
C02384=1053.098,186.427,409.804,171.634,34.791,156.522
C02385=1053.103,186.676,409.779,171.636,34.793,156.523
C02386=1053.110,186.925,409.755,171.638,34.796,156.523
C02387=1053.115,187.174,409.732,171.641,34.798,156.524
C02388=1053.121,187.422,409.708,171.643,34.801,156.524
C02389=1053.127,187.672,409.684,171.645,34.804,156.525
C02390=1053.133,187.920,409.660,171.648,34.806,156.525
C02391=1053.139,188.168,409.636,171.650,34.809,156.526
C02392=1053.145,188.418,409.612,171.652,34.811,156.526
C02393=1053.151,188.667,409.589,171.654,34.814,156.527
C02394=1053.156,188.916,409.564,171.657,34.817,156.527
C02395=1053.163,189.164,409.540,171.659,34.819,156.528
C02396=1053.168,189.413,409.516,171.661,34.822,156.528
C02397=1053.174,189.662,409.492,171.663,34.825,156.529
C02398=1053.181,189.946,409.465,171.666,34.827,156.529
C02399=1053.188,190.229,409.437,171.668,34.830,156.530
C02400=1053.194,190.514,409.409,171.672,34.834,156.530
C02401=1053.201,190.798,409.382,171.674,34.837,156.531
C02402=1053.207,191.047,409.358,171.676,34.839,156.531
C02403=1053.212,191.296,409.334,171.678,34.842,156.532
C02404=1053.218,191.544,409.310,171.681,34.845,156.532
C02405=1053.224,191.794,409.286,171.683,34.847,156.533
C02406=1053.230,192.042,409.262,171.686,34.850,156.533
C02407=1053.236,192.291,409.238,171.688,34.853,156.534
C02408=1053.242,192.540,409.214,171.690,34.855,156.534
C02409=1053.248,192.789,409.189,171.692,34.858,156.535
C02410=1053.254,193.037,409.166,171.695,34.860,156.535
C02411=1053.260,193.286,409.141,171.697,34.863,156.536
C02412=1053.266,193.534,409.117,171.700,34.866,156.536
C02413=1053.272,193.783,409.092,171.702,34.868,156.537
C02414=1053.278,194.032,409.068,171.704,34.871,156.537
C02415=1053.284,194.281,409.044,171.706,34.874,156.538
C02416=1053.290,194.529,409.020,171.709,34.876,156.538
C02417=1053.296,194.779,408.995,171.711,34.879,156.539
C02418=1053.302,195.027,408.972,171.714,34.882,156.539
C02419=1053.308,195.276,408.947,171.716,34.885,156.540
C02420=1053.314,195.524,408.924,171.718,34.887,156.540
C02421=1053.320,195.774,408.899,171.721,34.890,156.541
C02422=1053.327,196.022,408.874,171.723,34.893,156.541
C02423=1053.332,196.271,408.850,171.725,34.895,156.542
C02424=1053.338,196.520,408.825,171.728,34.898,156.542
C02425=1053.344,196.768,408.802,171.730,34.901,156.543
C02426=1053.350,197.017,408.777,171.733,34.903,156.543
C02427=1053.357,197.266,408.752,171.735,34.906,156.544
C02428=1053.362,197.514,408.728,171.737,34.909,156.544
C02429=1053.369,197.763,408.704,171.739,34.911,156.545
C02430=1053.374,198.012,408.680,171.743,34.914,156.545
C02431=1053.381,198.261,408.654,171.745,34.917,156.546
C02432=1053.387,198.510,408.630,171.747,34.919,156.546
C02433=1053.393,198.758,408.606,171.749,34.922,156.547
C02434=1053.399,199.007,408.582,171.752,34.925,156.547
C02435=1053.405,199.256,408.557,171.754,34.927,156.548
C02436=1053.411,199.504,408.533,171.757,34.930,156.548
C02437=1053.417,199.753,408.508,171.759,34.933,156.549
C02438=1053.423,200.001,408.483,171.761,34.935,156.549
C02439=1053.430,200.250,408.459,171.764,34.938,156.550
C02440=1053.435,200.500,408.435,171.766,34.941,156.550
C02441=1053.442,200.748,408.410,171.768,34.943,156.551
C02442=1053.448,200.997,408.386,171.772,34.946,156.551
C02443=1053.454,201.246,408.361,171.774,34.949,156.552
C02444=1053.461,201.494,408.336,171.776,34.952,156.552
C02445=1053.466,201.743,408.312,171.778,34.954,156.553
C02446=1053.472,201.991,408.287,171.781,34.957,156.553
C02447=1053.478,202.241,408.262,171.783,34.960,156.554
C02448=1053.484,202.488,408.238,171.786,34.963,156.554
C02449=1053.490,202.738,408.213,171.788,34.965,156.555
C02450=1053.496,202.986,408.188,171.791,34.968,156.555
C02451=1053.502,203.235,408.164,171.793,34.971,156.556
C02452=1053.508,203.484,408.138,171.795,34.974,156.556
C02453=1053.514,203.733,408.114,171.798,34.977,156.557
C02454=1053.519,203.981,408.089,171.801,34.979,156.557
C02455=1053.525,204.230,408.064,171.803,34.982,156.558
C02456=1053.532,204.479,408.039,171.805,34.985,156.558
C02457=1053.538,204.727,408.014,171.807,34.988,156.559
C02458=1053.544,204.976,407.990,171.810,34.991,156.560
C02459=1053.550,205.224,407.964,171.813,34.994,156.560
C02460=1053.556,205.473,407.939,171.815,34.997,156.561
C02461=1053.561,205.722,407.915,171.818,34.999,156.561
C02462=1053.587,206.773,407.809,172.030,35.092,156.577
C02463=1053.594,207.017,407.784,172.033,35.096,156.578
C02464=1053.599,207.260,407.758,172.034,35.100,156.578
C02465=1053.606,207.504,407.733,172.036,35.103,156.579
C02466=1053.612,207.747,407.707,172.038,35.106,156.580
C02467=1053.618,207.991,407.682,172.040,35.110,156.580
C02468=1053.624,208.235,407.656,172.042,35.113,156.581
C02469=1053.630,208.478,407.632,172.044,35.117,156.582
C02470=1053.637,208.722,407.606,172.045,35.121,156.582
C02471=1053.643,208.971,407.580,172.048,35.124,156.583
C02472=1053.649,209.219,407.554,172.050,35.128,156.584
C02473=1053.656,209.467,407.527,172.052,35.132,156.585
C02474=1053.662,209.716,407.501,172.054,35.135,156.585
C02475=1053.668,209.965,407.475,172.056,35.139,156.586
C02476=1053.675,210.213,407.450,172.058,35.142,156.587
C02477=1053.681,210.462,407.423,172.059,35.146,156.587
C02478=1053.687,210.710,407.397,172.062,35.150,156.588
C02479=1053.694,210.959,407.372,172.064,35.153,156.589
C02480=1053.700,211.208,407.345,172.065,35.157,156.590
C02481=1053.707,211.456,407.319,172.067,35.160,156.590
C02482=1053.713,211.705,407.293,172.070,35.164,156.591
C02483=1053.719,211.953,407.267,172.072,35.168,156.592
C02484=1053.726,212.202,407.240,172.073,35.171,156.593
C02485=1053.731,212.450,407.213,172.076,35.175,156.593
C02486=1053.738,212.699,407.188,172.078,35.179,156.594
C02487=1053.744,212.948,407.161,172.080,35.182,156.595
C02488=1053.751,213.196,407.135,172.081,35.186,156.595
C02489=1053.756,213.444,407.108,172.084,35.189,156.596
C02490=1053.763,213.693,407.082,172.086,35.193,156.597
C02491=1053.769,213.942,407.056,172.088,35.197,156.598
C02492=1053.775,214.190,407.030,172.090,35.200,156.598
C02493=1053.781,214.438,407.003,172.092,35.204,156.599
C02494=1053.788,214.687,406.977,172.094,35.207,156.600
C02495=1053.794,214.936,406.950,172.096,35.211,156.600
C02496=1053.801,215.184,406.924,172.098,35.215,156.601
C02497=1053.807,215.433,406.897,172.100,35.218,156.602
C02498=1053.813,215.681,406.871,172.102,35.222,156.603
C02499=1053.820,215.930,406.845,172.105,35.226,156.603
C02500=1053.825,216.179,406.818,172.106,35.229,156.604
C02501=1053.832,216.427,406.792,172.108,35.233,156.605
C02502=1053.838,216.676,406.765,172.110,35.236,156.605
C02503=1053.845,216.924,406.739,172.113,35.240,156.606
C02504=1053.850,217.172,406.712,172.114,35.244,156.607
C02505=1053.858,217.421,406.686,172.116,35.247,156.608
C02506=1053.863,217.669,406.659,172.119,35.251,156.608
C02507=1053.870,217.918,406.632,172.121,35.254,156.609
C02508=1053.876,218.167,406.606,172.123,35.258,156.610
C02509=1053.882,218.415,406.580,172.124,35.262,156.611
C02510=1053.889,218.664,406.553,172.127,35.265,156.611
C02511=1053.895,218.912,406.527,172.129,35.268,156.612
C02512=1053.902,219.161,406.500,172.131,35.272,156.613
C02513=1053.908,219.409,406.474,172.134,35.276,156.613
C02514=1053.914,219.658,406.447,172.135,35.279,156.614
C02515=1053.921,219.906,406.420,172.137,35.283,156.615
C02516=1053.927,220.155,406.393,172.139,35.286,156.615
C02517=1053.934,220.403,406.367,172.142,35.290,156.616
C02518=1053.940,220.652,406.340,172.144,35.294,156.617
C02519=1053.946,220.898,406.314,172.146,35.297,156.618
C02520=1053.952,221.144,406.287,172.148,35.300,156.618
C02521=1053.959,221.391,406.260,172.150,35.304,156.619
C02522=1053.964,221.637,406.234,172.152,35.307,156.620
C02523=1053.971,221.883,406.207,172.154,35.311,156.620
C02524=1053.977,222.129,406.181,172.157,35.315,156.621
C02525=1053.984,222.375,406.153,172.158,35.318,156.622
C02526=1053.989,222.621,406.127,172.160,35.322,156.623
C02527=1053.996,222.870,406.100,172.163,35.325,156.623
C02528=1054.002,223.118,406.074,172.165,35.329,156.624
C02529=1054.009,223.367,406.047,172.167,35.333,156.625
C02530=1054.014,223.615,406.020,172.168,35.336,156.625
C02531=1054.021,223.864,405.993,172.171,35.340,156.626
C02532=1054.027,224.112,405.966,172.173,35.343,156.627
C02533=1054.033,224.361,405.939,172.175,35.346,156.628
C02534=1054.039,224.610,405.912,172.178,35.350,156.628
C02535=1054.047,224.858,405.885,172.180,35.354,156.629
C02536=1054.052,225.106,405.858,172.182,35.357,156.630
C02537=1054.059,225.355,405.831,172.184,35.361,156.630
C02538=1054.065,225.603,405.804,172.186,35.364,156.631
C02539=1054.071,225.852,405.777,172.188,35.368,156.632
C02540=1054.077,226.100,405.749,172.190,35.372,156.633
C02541=1054.084,226.349,405.722,172.193,35.375,156.633
C02542=1054.091,226.597,405.696,172.195,35.379,156.634
C02543=1054.097,226.845,405.669,172.197,35.382,156.635
C02544=1054.103,227.094,405.642,172.200,35.385,156.635
C02545=1054.109,227.342,405.614,172.201,35.389,156.636
C02546=1054.116,227.591,405.587,172.203,35.393,156.637
C02547=1054.121,227.839,405.561,172.206,35.396,156.638
C02548=1054.128,228.088,405.533,172.208,35.400,156.638
C02549=1054.134,228.337,405.506,172.210,35.403,156.639
C02550=1054.141,228.584,405.479,172.212,35.406,156.640
C02551=1054.148,228.833,405.452,172.215,35.410,156.640
C02552=1054.154,229.082,405.424,172.217,35.414,156.641
C02553=1054.160,229.330,405.398,172.219,35.417,156.642
C02554=1054.167,229.579,405.370,172.222,35.421,156.642
C02555=1054.173,229.826,405.343,172.224,35.424,156.643
C02556=1054.179,230.075,405.316,172.225,35.428,156.644
C02557=1054.185,230.324,405.287,172.228,35.432,156.645
C02558=1054.191,230.573,405.261,172.230,35.435,156.645
C02559=1054.198,230.821,405.233,172.232,35.438,156.646
C02560=1054.204,231.069,405.205,172.234,35.442,156.647
C02561=1054.210,231.318,405.178,172.237,35.445,156.647
C02562=1054.217,231.566,405.151,172.239,35.449,156.648
C02563=1054.223,231.814,405.123,172.241,35.453,156.649
C02564=1054.229,232.063,405.096,172.244,35.456,156.650
C02565=1054.236,232.311,405.069,172.246,35.460,156.650
C02566=1054.242,232.559,405.041,172.248,35.463,156.651
C02567=1054.248,232.809,405.014,172.251,35.466,156.652
C02568=1054.254,233.057,404.986,172.253,35.470,156.652
C02569=1054.260,233.305,404.959,172.254,35.474,156.653
C02570=1054.267,233.553,404.931,172.257,35.477,156.654
C02571=1054.273,233.802,404.903,172.259,35.481,156.655
C02572=1054.279,234.050,404.876,172.261,35.484,156.655
C02573=1054.285,234.299,404.848,172.264,35.488,156.656
C02574=1054.292,234.547,404.820,172.266,35.492,156.657
C02575=1054.298,234.790,404.794,172.268,35.495,156.657
C02576=1054.304,235.032,404.767,172.270,35.498,156.658
C02577=1054.310,235.274,404.740,172.273,35.502,156.659
C02578=1054.316,235.517,404.713,172.275,35.505,156.660
C02579=1054.322,235.759,404.686,172.277,35.508,156.660
C02580=1054.328,236.001,404.658,172.280,35.512,156.661
C02581=1054.334,236.243,404.631,172.282,35.516,156.662
C02582=1054.340,236.486,404.604,172.284,35.519,156.662
C02583=1054.347,236.734,404.577,172.287,35.522,156.663
C02584=1054.354,236.983,404.549,172.289,35.526,156.664
C02585=1054.360,237.231,404.521,172.291,35.529,156.664
C02586=1054.366,237.479,404.493,172.294,35.533,156.665
C02587=1054.372,237.728,404.465,172.296,35.536,156.666
C02588=1054.379,237.976,404.438,172.298,35.540,156.667
C02589=1054.385,238.225,404.409,172.300,35.543,156.667
C02590=1054.391,238.473,404.382,172.303,35.547,156.668
C02591=1054.398,238.721,404.354,172.305,35.550,156.669
C02592=1054.405,238.969,404.327,172.307,35.554,156.669
C02593=1054.410,239.218,404.298,172.310,35.557,156.670
C02594=1054.417,239.467,404.270,172.312,35.561,156.671
C02595=1054.422,239.715,404.242,172.314,35.565,156.672
C02596=1054.429,239.963,404.215,172.317,35.568,156.672
C02597=1054.436,240.212,404.187,172.319,35.571,156.673
C02598=1054.442,240.460,404.159,172.321,35.575,156.674
C02599=1054.448,240.709,404.131,172.324,35.578,156.674
C02600=1054.455,240.957,404.103,172.326,35.582,156.675
C02601=1054.460,241.205,404.075,172.328,35.585,156.676
C02602=1054.467,241.453,404.047,172.331,35.588,156.676
C02603=1054.474,241.702,404.019,172.333,35.592,156.677
C02604=1054.480,241.950,403.991,172.335,35.596,156.678
C02605=1054.487,242.199,403.963,172.338,35.599,156.679
C02606=1054.493,242.447,403.935,172.340,35.603,156.679
C02607=1054.498,242.696,403.907,172.342,35.606,156.680
C02608=1054.505,242.943,403.878,172.345,35.610,156.681
C02609=1054.511,243.192,403.850,172.347,35.613,156.681
C02610=1054.518,243.441,403.822,172.349,35.616,156.682
C02611=1054.524,243.689,403.793,172.352,35.620,156.683
C02612=1054.531,243.937,403.765,172.354,35.624,156.684
C02613=1054.537,244.186,403.737,172.356,35.627,156.684
C02614=1054.542,244.434,403.709,172.359,35.631,156.685
C02615=1054.549,244.682,403.681,172.361,35.634,156.686
C02616=1054.555,244.930,403.652,172.363,35.638,156.687
C02617=1054.562,245.178,403.624,172.367,35.641,156.687
C02618=1054.568,245.427,403.596,172.369,35.645,156.688
C02619=1054.574,245.676,403.567,172.371,35.648,156.689
C02620=1054.581,245.924,403.539,172.374,35.652,156.689
C02621=1054.587,246.172,403.511,172.376,35.655,156.690
C02622=1054.593,246.421,403.482,172.378,35.659,156.691
C02623=1054.598,246.669,403.454,172.381,35.662,156.692
C02624=1054.605,246.917,403.426,172.383,35.666,156.692
C02625=1054.611,247.165,403.397,172.385,35.670,156.693
C02626=1054.617,247.414,403.368,172.388,35.673,156.694
C02627=1054.623,247.662,403.339,172.390,35.677,156.695
C02628=1054.629,247.911,403.311,172.392,35.680,156.695
C02629=1054.636,248.159,403.283,172.396,35.684,156.696
C02630=1054.643,248.407,403.254,172.398,35.687,156.697
C02631=1054.648,248.646,403.226,172.400,35.690,156.697
C02632=1054.654,248.886,403.199,172.403,35.694,156.698
C02633=1054.660,249.125,403.171,172.405,35.698,156.699
C02634=1054.666,249.365,403.143,172.407,35.701,156.700
C02635=1054.672,249.603,403.116,172.410,35.704,156.700
C02636=1054.678,249.843,403.088,172.412,35.708,156.701
C02637=1054.684,250.082,403.061,172.414,35.711,156.702
C02638=1054.690,250.321,403.033,172.417,35.714,156.702
C02639=1054.696,250.570,403.005,172.419,35.718,156.703
C02640=1054.702,250.818,402.976,172.421,35.721,156.704
C02641=1054.708,251.066,402.946,172.424,35.725,156.705
C02642=1054.715,251.314,402.918,172.426,35.728,156.705
C02643=1054.721,251.563,402.890,172.429,35.732,156.706
C02644=1054.727,251.811,402.861,172.432,35.736,156.707
C02645=1054.734,252.059,402.832,172.434,35.739,156.707
C02646=1054.740,252.308,402.803,172.436,35.743,156.708
C02647=1054.746,252.556,402.774,172.439,35.746,156.709
C02648=1054.752,252.804,402.745,172.441,35.749,156.710
C02649=1054.758,253.052,402.716,172.443,35.753,156.710
C02650=1054.765,253.301,402.688,172.447,35.756,156.711
C02651=1054.771,253.549,402.659,172.449,35.760,156.712
C02652=1054.777,253.797,402.630,172.451,35.764,156.712
C02653=1054.784,254.045,402.601,172.454,35.767,156.713
C02654=1054.790,254.293,402.572,172.456,35.771,156.714
C02655=1054.797,254.542,402.543,172.459,35.774,156.715
C02656=1054.803,254.791,402.515,172.462,35.777,156.715
C02657=1054.809,255.039,402.486,172.464,35.781,156.716
C02658=1054.815,255.287,402.456,172.467,35.784,156.717
C02659=1054.821,255.535,402.427,172.469,35.788,156.718
C02660=1054.828,255.783,402.399,172.471,35.791,156.718
C02661=1054.835,256.031,402.370,172.475,35.795,156.719
C02662=1054.841,256.279,402.341,172.477,35.799,156.720
C02663=1054.847,256.528,402.312,172.479,35.802,156.720
C02664=1054.854,256.776,402.282,172.482,35.805,156.721
C02665=1054.860,257.025,402.253,172.484,35.809,156.722
C02666=1054.867,257.273,402.224,172.487,35.812,156.723
C02667=1054.873,257.521,402.195,172.490,35.816,156.723
C02668=1054.879,257.769,402.166,172.492,35.819,156.724
C02669=1054.885,258.017,402.137,172.494,35.822,156.725
C02670=1054.892,258.266,402.108,172.498,35.826,156.725
C02671=1054.898,258.514,402.079,172.500,35.829,156.726
C02672=1054.905,258.762,402.050,172.502,35.833,156.727
C02673=1054.911,259.010,402.021,172.505,35.837,156.728
C02674=1054.917,259.258,401.992,172.507,35.840,156.728
C02675=1054.924,259.507,401.962,172.511,35.843,156.729
C02676=1054.931,259.755,401.934,172.513,35.847,156.730
C02677=1054.937,260.003,401.905,172.515,35.850,156.730
C02678=1054.944,260.251,401.876,172.519,35.854,156.731
C02679=1054.951,260.500,401.846,172.521,35.857,156.732
C02680=1054.957,260.748,401.817,172.523,35.861,156.733
C02681=1054.963,260.996,401.788,172.526,35.864,156.733
C02682=1054.969,261.244,401.759,172.529,35.867,156.734
C02683=1054.976,261.493,401.729,172.531,35.871,156.735
C02684=1054.983,261.741,401.700,172.534,35.874,156.736
C02685=1054.989,261.988,401.670,172.536,35.878,156.736
C02686=1054.996,262.237,401.641,172.539,35.881,156.737
C02687=1055.001,262.476,401.613,172.542,35.885,156.738
C02688=1055.008,262.714,401.585,172.544,35.888,156.738
C02689=1055.015,262.953,401.557,172.546,35.891,156.739
C02690=1055.021,263.191,401.528,172.550,35.895,156.740
C02691=1055.026,263.429,401.500,172.552,35.898,156.740
C02692=1055.032,263.668,401.471,172.555,35.901,156.741
C02693=1055.039,263.906,401.443,172.557,35.905,156.742
C02694=1055.044,264.144,401.415,172.559,35.908,156.743
C02695=1055.051,264.392,401.385,172.563,35.912,156.743
C02696=1055.057,264.641,401.355,172.565,35.915,156.744
C02697=1055.063,264.888,401.325,172.567,35.919,156.745
C02698=1055.070,265.137,401.296,172.570,35.922,156.746
C02699=1055.076,265.386,401.266,172.573,35.925,156.746
C02700=1055.082,265.633,401.236,172.575,35.929,156.747
C02701=1055.088,265.881,401.207,172.578,35.932,156.748
C02702=1055.095,266.130,401.177,172.581,35.936,156.748
C02703=1055.101,266.378,401.148,172.584,35.940,156.749
C02704=1055.108,266.625,401.118,172.586,35.943,156.750
C02705=1055.114,266.875,401.088,172.589,35.947,156.751
C02706=1055.120,267.122,401.058,172.592,35.950,156.751
C02707=1055.127,267.370,401.028,172.594,35.954,156.752
C02708=1055.133,267.619,400.998,172.598,35.957,156.753
C02709=1055.140,267.866,400.969,172.600,35.961,156.754
C02710=1055.146,268.114,400.940,172.602,35.964,156.754
C02711=1055.152,268.363,400.909,172.606,35.968,156.755
C02712=1055.159,268.610,400.879,172.608,35.971,156.756
C02713=1055.165,268.860,400.849,172.610,35.975,156.757
C02714=1055.171,269.107,400.819,172.614,35.979,156.757
C02715=1055.177,269.355,400.789,172.616,35.982,156.758
C02716=1055.184,269.604,400.760,172.619,35.986,156.759
C02717=1055.190,269.852,400.729,172.622,35.989,156.760
C02718=1055.196,270.099,400.700,172.624,35.993,156.760
C02719=1055.203,270.348,400.670,172.627,35.996,156.761
C02720=1055.209,270.596,400.640,172.630,36.000,156.762
C02721=1055.216,270.844,400.609,172.633,36.003,156.763
C02722=1055.222,271.092,400.579,172.635,36.007,156.763
C02723=1055.228,271.340,400.550,172.638,36.010,156.764
C02724=1055.235,271.588,400.520,172.641,36.014,156.765
C02725=1055.241,271.836,400.489,172.644,36.017,156.766
C02726=1055.248,272.084,400.459,172.646,36.021,156.766
C02727=1055.254,272.332,400.429,172.649,36.024,156.767
C02728=1055.261,272.580,400.399,172.652,36.028,156.768
C02729=1055.266,272.829,400.369,172.655,36.032,156.769
C02730=1055.273,273.077,400.338,172.658,36.035,156.769
C02731=1055.279,273.325,400.308,172.660,36.039,156.770
C02732=1055.285,273.573,400.278,172.663,36.042,156.771
C02733=1055.291,273.821,400.247,172.666,36.046,156.772
C02734=1055.298,274.069,400.218,172.669,36.049,156.772
C02735=1055.304,274.317,400.187,172.672,36.053,156.773
C02736=1055.310,274.565,400.157,172.674,36.056,156.774
C02737=1055.317,274.813,400.126,172.677,36.060,156.775
C02738=1055.323,275.061,400.096,172.680,36.063,156.775
C02739=1055.330,275.310,400.065,172.683,36.067,156.776
C02740=1055.336,275.557,400.036,172.686,36.070,156.777
C02741=1055.343,275.806,400.005,172.688,36.074,156.778
C02742=1055.348,276.054,399.975,172.691,36.077,156.778
C02743=1055.355,276.294,399.945,172.694,36.081,156.779
C02744=1055.361,276.535,399.915,172.697,36.084,156.780
C02745=1055.367,276.775,399.885,172.700,36.088,156.781
C02746=1055.374,277.015,399.856,172.702,36.092,156.781
C02747=1055.380,277.255,399.827,172.705,36.095,156.782
C02748=1055.386,277.496,399.798,172.708,36.099,156.783
C02749=1055.392,277.736,399.767,172.711,36.102,156.784
C02750=1055.398,277.976,399.738,172.713,36.106,156.784
C02751=1055.405,278.225,399.707,172.716,36.109,156.785
C02752=1055.411,278.473,399.677,172.719,36.113,156.786
C02753=1055.417,278.721,399.646,172.722,36.116,156.787
C02754=1055.424,278.969,399.615,172.725,36.120,156.787
C02755=1055.430,279.217,399.585,172.728,36.123,156.788
C02756=1055.437,279.465,399.554,172.730,36.127,156.789
C02757=1055.443,279.713,399.523,172.734,36.130,156.790
C02758=1055.449,279.961,399.493,172.736,36.134,156.790
C02759=1055.455,280.209,399.462,172.740,36.138,156.791
C02760=1055.462,280.457,399.431,172.742,36.141,156.792
C02761=1055.468,280.705,399.400,172.745,36.145,156.793
C02762=1055.474,280.954,399.369,172.748,36.148,156.793
C02763=1055.481,281.201,399.338,172.750,36.152,156.794
C02764=1055.487,281.449,399.308,172.754,36.155,156.795
C02765=1055.493,281.697,399.277,172.756,36.160,156.796
C02766=1055.500,281.945,399.246,172.760,36.163,156.797
C02767=1055.506,282.194,399.215,172.762,36.167,156.797
C02768=1055.512,282.441,399.184,172.765,36.170,156.798
C02769=1055.518,282.689,399.153,172.768,36.174,156.799
C02770=1055.525,282.937,399.122,172.771,36.178,156.800
C02771=1055.531,283.185,399.092,172.774,36.181,156.800
C02772=1055.538,283.433,399.060,172.777,36.185,156.801
C02773=1055.544,283.681,399.029,172.780,36.188,156.802
C02774=1055.550,283.929,398.998,172.783,36.192,156.803
C02775=1055.557,284.177,398.967,172.786,36.196,156.804
C02776=1055.563,284.425,398.936,172.789,36.199,156.804
C02777=1055.570,284.672,398.905,172.792,36.203,156.805
C02778=1055.576,284.921,398.874,172.795,36.206,156.806
C02779=1055.583,285.169,398.843,172.798,36.210,156.807
C02780=1055.589,285.416,398.812,172.801,36.214,156.807
C02781=1055.595,285.664,398.781,172.804,36.217,156.808
C02782=1055.602,285.912,398.750,172.806,36.221,156.809
C02783=1055.609,286.160,398.718,172.810,36.224,156.810
C02784=1055.615,286.408,398.688,172.812,36.228,156.810
C02785=1055.621,286.656,398.657,172.816,36.231,156.811
C02786=1055.628,286.904,398.625,172.819,36.236,156.812
C02787=1055.634,287.152,398.594,172.822,36.239,156.813
C02788=1055.641,287.400,398.563,172.825,36.243,156.814
C02789=1055.647,287.647,398.532,172.827,36.246,156.814
C02790=1055.654,287.895,398.500,172.831,36.250,156.815
C02791=1055.660,288.144,398.468,172.833,36.254,156.816
C02792=1055.666,288.392,398.438,172.837,36.257,156.817
C02793=1055.673,288.640,398.406,172.840,36.261,156.818
C02794=1055.679,288.887,398.375,172.843,36.265,156.818
C02795=1055.685,289.135,398.343,172.846,36.268,156.819
C02796=1055.692,289.383,398.312,172.849,36.272,156.820
C02797=1055.699,289.631,398.280,172.852,36.276,156.821
C02798=1055.705,289.879,398.249,172.855,36.279,156.822
C02799=1055.711,290.125,398.217,172.858,36.283,156.822
C02800=1055.718,290.371,398.187,172.861,36.286,156.823
C02801=1055.724,290.616,398.155,172.864,36.290,156.824
C02802=1055.731,290.863,398.124,172.867,36.294,156.825
C02803=1055.737,291.109,398.093,172.870,36.297,156.825
C02804=1055.742,291.354,398.061,172.873,36.301,156.826
C02805=1055.750,291.601,398.030,172.877,36.305,156.827
C02806=1055.755,291.846,397.999,172.879,36.308,156.828
C02807=1055.762,292.094,397.967,172.882,36.312,156.829
C02808=1055.769,292.342,397.936,172.886,36.316,156.830
C02809=1055.775,292.590,397.904,172.888,36.320,156.830
C02810=1055.781,292.838,397.873,172.892,36.324,156.831
C02811=1055.788,293.085,397.841,172.894,36.327,156.832
C02812=1055.794,293.333,397.809,172.898,36.331,156.833
C02813=1055.801,293.581,397.777,172.901,36.335,156.834
C02814=1055.807,293.829,397.745,172.904,36.338,156.834
C02815=1055.813,294.077,397.714,172.907,36.342,156.835
C02816=1055.820,294.325,397.682,172.911,36.346,156.836
C02817=1055.826,294.573,397.649,172.913,36.349,156.837
C02818=1055.833,294.821,397.618,172.917,36.353,156.838
C02819=1055.839,295.069,397.586,172.920,36.357,156.838
C02820=1055.846,295.317,397.555,172.922,36.360,156.839
C02821=1055.852,295.564,397.522,172.926,36.364,156.840
C02822=1055.859,295.812,397.490,172.929,36.368,156.841
C02823=1055.865,296.060,397.458,172.932,36.372,156.842
C02824=1055.872,296.308,397.426,172.935,36.375,156.842
C02825=1055.878,296.556,397.394,172.939,36.379,156.843
C02826=1055.885,296.804,397.363,172.941,36.383,156.844
C02827=1055.890,297.051,397.330,172.945,36.387,156.845
C02828=1055.896,297.299,397.298,172.948,36.390,156.846
C02829=1055.903,297.547,397.266,172.951,36.394,156.847
C02830=1055.909,297.794,397.234,172.954,36.399,156.848
C02831=1055.916,298.042,397.201,172.958,36.402,156.848
C02832=1055.922,298.290,397.169,172.960,36.406,156.849
C02833=1055.928,298.538,397.137,172.964,36.410,156.850
C02834=1055.935,298.786,397.105,172.967,36.414,156.851
C02835=1055.941,299.033,397.072,172.971,36.418,156.852
C02836=1055.947,299.282,397.040,172.973,36.421,156.853
C02837=1055.953,299.529,397.008,172.977,36.425,156.853
C02838=1055.959,299.777,396.976,172.980,36.429,156.854
C02839=1055.966,300.025,396.944,172.983,36.433,156.855
C02840=1055.973,300.272,396.911,172.986,36.437,156.856
C02841=1055.979,300.520,396.879,172.990,36.441,156.857
C02842=1055.985,300.768,396.846,172.993,36.444,156.858
C02843=1055.992,301.015,396.814,172.996,36.448,156.858
C02844=1055.998,301.264,396.782,172.999,36.452,156.859
C02845=1056.004,301.511,396.749,173.003,36.456,156.860
C02846=1056.010,301.759,396.716,173.006,36.460,156.861
C02847=1056.016,302.007,396.684,173.009,36.463,156.862
C02848=1056.023,302.254,396.652,173.012,36.467,156.863
C02849=1056.030,302.502,396.619,173.016,36.471,156.864
C02850=1056.037,302.750,396.586,173.019,36.475,156.864
C02851=1056.043,302.998,396.554,173.022,36.479,156.865
C02852=1056.049,303.246,396.522,173.025,36.483,156.866
C02853=1056.055,303.493,396.489,173.029,36.487,156.867
C02854=1056.062,303.741,396.456,173.032,36.491,156.868
C02855=1056.068,304.000,396.422,173.036,36.495,156.869
C02856=1056.076,304.260,396.388,173.038,36.499,156.870
C02857=1056.082,304.519,396.354,173.042,36.503,156.870
C02858=1056.089,304.780,396.320,173.045,36.507,156.871
C02859=1056.095,305.028,396.287,173.049,36.511,156.872
C02860=1056.102,305.275,396.255,173.052,36.515,156.873
C02861=1056.109,305.523,396.222,173.056,36.518,156.874
C02862=1056.115,305.770,396.189,173.059,36.522,156.875
C02863=1056.122,306.019,396.156,173.062,36.526,156.876
C02864=1056.128,306.266,396.123,173.065,36.530,156.877
C02865=1056.134,306.514,396.091,173.069,36.534,156.877
C02866=1056.141,306.761,396.058,173.072,36.538,156.878
C02867=1056.147,307.010,396.025,173.076,36.542,156.879
C02868=1056.154,307.257,395.993,173.079,36.545,156.880
C02869=1056.161,307.504,395.960,173.082,36.549,156.881
C02870=1056.167,307.752,395.927,173.085,36.553,156.882
C02871=1056.174,308.000,395.893,173.089,36.557,156.883
C02872=1056.181,308.247,395.861,173.092,36.561,156.883
C02873=1056.187,308.495,395.828,173.096,36.565,156.884
C02874=1056.194,308.743,395.795,173.100,36.569,156.885
C02875=1056.200,308.991,395.762,173.103,36.573,156.886
C02876=1056.206,309.238,395.729,173.106,36.576,156.887
C02877=1056.213,309.487,395.696,173.109,36.581,156.888
C02878=1056.221,309.733,395.663,173.113,36.585,156.889
C02879=1056.227,309.981,395.631,173.116,36.589,156.890
C02880=1056.234,310.229,395.597,173.120,36.593,156.890
C02881=1056.240,310.477,395.565,173.123,36.596,156.891
C02882=1056.247,310.724,395.531,173.127,36.600,156.892
C02883=1056.254,310.972,395.498,173.130,36.604,156.893
C02884=1056.260,311.220,395.465,173.134,36.608,156.894
C02885=1056.267,311.467,395.432,173.136,36.612,156.895
C02886=1056.273,311.715,395.399,173.140,36.616,156.896
C02887=1056.280,311.963,395.366,173.143,36.620,156.897
C02888=1056.287,312.210,395.332,173.147,36.624,156.897
C02889=1056.293,312.458,395.300,173.150,36.628,156.898
C02890=1056.300,312.706,395.266,173.154,36.632,156.899
C02891=1056.307,312.953,395.233,173.158,36.636,156.900
C02892=1056.314,313.201,395.200,173.161,36.639,156.901
C02893=1056.320,313.450,395.167,173.165,36.643,156.902
C02894=1056.327,313.697,395.133,173.168,36.647,156.903
C02895=1056.333,313.944,395.099,173.172,36.651,156.904
C02896=1056.340,314.192,395.066,173.174,36.656,156.905
C02897=1056.346,314.439,395.032,173.178,36.660,156.906
C02898=1056.352,314.687,394.999,173.181,36.664,156.906
C02899=1056.359,314.935,394.966,173.185,36.668,156.907
C02900=1056.365,315.182,394.931,173.189,36.672,156.908
C02901=1056.372,315.430,394.898,173.192,36.676,156.909
C02902=1056.378,315.678,394.864,173.196,36.680,156.910
C02903=1056.385,315.925,394.830,173.199,36.684,156.911
C02904=1056.390,316.173,394.797,173.203,36.688,156.912
C02905=1056.397,316.420,394.764,173.206,36.692,156.913
C02906=1056.404,316.668,394.729,173.210,36.696,156.914
C02907=1056.410,316.915,394.696,173.214,36.700,156.915
C02908=1056.416,317.164,394.662,173.217,36.705,156.916
C02909=1056.423,317.411,394.629,173.221,36.709,156.917
C02910=1056.429,317.659,394.594,173.223,36.713,156.918
C02911=1056.438,317.971,394.551,173.228,36.718,156.919
C02912=1056.445,318.283,394.509,173.233,36.723,156.920
C02913=1056.453,318.595,394.466,173.238,36.728,156.921
C02914=1056.462,318.908,394.424,173.241,36.734,156.922
C02915=1056.469,319.156,394.390,173.245,36.738,156.923
C02916=1056.475,319.403,394.356,173.249,36.742,156.924
C02917=1056.482,319.651,394.322,173.252,36.746,156.925
C02918=1056.488,319.898,394.288,173.256,36.751,156.926
C02919=1056.495,320.146,394.254,173.259,36.755,156.927
C02920=1056.501,320.394,394.220,173.263,36.759,156.928
C02921=1056.508,320.640,394.186,173.266,36.763,156.929
C02922=1056.514,320.888,394.152,173.270,36.767,156.930
C02923=1056.522,321.136,394.118,173.274,36.771,156.931
C02924=1056.528,321.383,394.084,173.277,36.775,156.932
C02925=1056.534,321.631,394.050,173.282,36.780,156.933
C02926=1056.541,321.879,394.016,173.286,36.784,156.934
C02927=1056.547,322.126,393.982,173.289,36.788,156.935
C02928=1056.555,322.373,393.947,173.293,36.792,156.936
C02929=1056.561,322.621,393.913,173.296,36.796,156.936
C02930=1056.568,322.868,393.879,173.300,36.800,156.937
C02931=1056.574,323.116,393.845,173.304,36.805,156.938
C02932=1056.581,323.364,393.810,173.307,36.809,156.939
C02933=1056.588,323.612,393.777,173.311,36.813,156.940
C02934=1056.594,323.859,393.743,173.314,36.817,156.941
C02935=1056.601,324.106,393.708,173.318,36.821,156.942
C02936=1056.608,324.354,393.674,173.322,36.826,156.943
C02937=1056.614,324.602,393.639,173.325,36.830,156.944
C02938=1056.621,324.849,393.606,173.329,36.834,156.945
C02939=1056.627,325.097,393.571,173.332,36.839,156.946
C02940=1056.635,325.344,393.537,173.336,36.843,156.947
C02941=1056.641,325.592,393.502,173.341,36.847,156.948
C02942=1056.648,325.840,393.467,173.344,36.851,156.949
C02943=1056.654,326.063,393.436,173.347,36.855,156.950
C02944=1056.660,326.286,393.405,173.351,36.859,156.951
C02945=1056.667,326.509,393.374,173.354,36.862,156.952
C02946=1056.672,326.733,393.343,173.358,36.866,156.952
C02947=1056.679,326.956,393.312,173.361,36.870,156.953
C02948=1056.684,327.180,393.281,173.365,36.874,156.954
C02949=1056.691,327.403,393.250,173.367,36.878,156.955
C02950=1056.697,327.626,393.218,173.371,36.882,156.956
C02951=1056.704,327.874,393.185,173.375,36.886,156.957
C02952=1056.711,328.121,393.149,173.378,36.890,156.958
C02953=1056.717,328.369,393.115,173.383,36.895,156.959
C02954=1056.725,328.616,393.080,173.386,36.899,156.960
C02955=1056.731,328.864,393.046,173.390,36.903,156.961
C02956=1056.738,329.112,393.011,173.394,36.907,156.962
C02957=1056.745,329.359,392.977,173.397,36.912,156.963
C02958=1056.751,329.606,392.942,173.401,36.916,156.964
C02959=1056.758,329.855,392.908,173.406,36.920,156.965
C02960=1056.766,330.102,392.873,173.409,36.925,156.966
C02961=1056.773,330.349,392.838,173.413,36.929,156.967
C02962=1056.778,330.596,392.804,173.417,36.933,156.968
C02963=1056.785,330.844,392.769,173.420,36.938,156.969
C02964=1056.792,331.091,392.734,173.424,36.942,156.970
C02965=1056.799,331.338,392.698,173.429,36.946,156.971
C02966=1056.805,331.586,392.663,173.432,36.951,156.972
C02967=1056.812,331.845,392.626,173.436,36.955,156.973
C02968=1056.819,332.103,392.590,173.440,36.960,156.974
C02969=1056.826,332.362,392.553,173.444,36.965,156.975
C02970=1056.833,332.620,392.517,173.448,36.970,156.976
C02971=1056.840,332.867,392.482,173.452,36.974,156.977
C02972=1056.847,333.115,392.447,173.457,36.979,156.978
C02973=1056.854,333.363,392.412,173.460,36.983,156.979
C02974=1056.861,333.610,392.376,173.464,36.988,156.980
C02975=1056.867,333.858,392.341,173.468,36.992,156.981
C02976=1056.873,334.105,392.306,173.471,36.996,156.982
C02977=1056.880,334.352,392.270,173.476,37.001,156.984
C02978=1056.887,334.600,392.235,173.480,37.005,156.985
C02979=1056.894,334.847,392.200,173.483,37.010,156.986
C02980=1056.900,335.095,392.165,173.487,37.014,156.987
C02981=1056.907,335.342,392.130,173.492,37.019,156.988
C02982=1056.914,335.589,392.095,173.495,37.023,156.989
C02983=1056.921,335.837,392.060,173.499,37.028,156.990
C02984=1056.928,336.084,392.023,173.503,37.032,156.991
C02985=1056.935,336.331,391.988,173.508,37.037,156.992
C02986=1056.941,336.579,391.953,173.511,37.041,156.993
C02987=1056.948,336.826,391.917,173.515,37.046,156.994
C02988=1056.955,337.074,391.882,173.519,37.050,156.995
C02989=1056.962,337.321,391.846,173.524,37.055,156.996
C02990=1056.968,337.568,391.811,173.527,37.060,156.997
C02991=1056.975,337.816,391.775,173.531,37.064,156.998
C02992=1056.982,338.063,391.739,173.536,37.069,156.999
C02993=1056.988,338.311,391.704,173.539,37.073,157.000
C02994=1056.995,338.558,391.668,173.543,37.078,157.002
C02995=1057.002,338.805,391.633,173.547,37.083,157.003
C02996=1057.009,339.053,391.597,173.552,37.087,157.004
C02997=1057.016,339.301,391.561,173.555,37.092,157.005
C02998=1057.023,339.547,391.526,173.559,37.096,157.006
C02999=1057.029,339.795,391.490,173.564,37.101,157.007
C03000=1057.036,340.042,391.454,173.568,37.106,157.008
C03001=1057.043,340.290,391.418,173.571,37.110,157.009
C03002=1057.049,340.537,391.382,173.576,37.116,157.010
C03003=1057.056,340.784,391.347,173.580,37.120,157.011
C03004=1057.064,341.032,391.311,173.584,37.125,157.013
C03005=1057.070,341.279,391.275,173.588,37.130,157.014
C03006=1057.077,341.526,391.239,173.592,37.134,157.015
C03007=1057.083,341.773,391.203,173.596,37.139,157.016
C03008=1057.091,342.021,391.167,173.601,37.144,157.017
C03009=1057.098,342.268,391.131,173.604,37.148,157.018
C03010=1057.105,342.516,391.094,173.609,37.153,157.019
C03011=1057.112,342.763,391.059,173.613,37.158,157.020
C03012=1057.119,343.010,391.023,173.617,37.162,157.021
C03013=1057.126,343.258,390.987,173.621,37.167,157.023
C03014=1057.132,343.505,390.951,173.625,37.172,157.024
C03015=1057.139,343.752,390.915,173.629,37.177,157.025
C03016=1057.146,344.000,390.878,173.634,37.181,157.026
C03017=1057.153,344.247,390.842,173.638,37.186,157.027
C03018=1057.159,344.494,390.806,173.642,37.191,157.028
C03019=1057.167,344.741,390.770,173.646,37.196,157.029
C03020=1057.173,344.989,390.734,173.650,37.201,157.031
C03021=1057.180,345.236,390.697,173.655,37.205,157.032
C03022=1057.187,345.483,390.661,173.658,37.210,157.033
C03023=1057.194,345.737,390.623,173.663,37.215,157.034
C03024=1057.201,345.992,390.586,173.667,37.220,157.035
C03025=1057.208,346.246,390.548,173.672,37.225,157.036
C03026=1057.215,346.499,390.512,173.676,37.230,157.038
C03027=1057.222,346.747,390.475,173.681,37.235,157.039
C03028=1057.228,346.994,390.439,173.684,37.240,157.040
C03029=1057.236,347.242,390.402,173.689,37.245,157.041
C03030=1057.242,347.489,390.366,173.693,37.250,157.042
C03031=1057.249,347.736,390.329,173.698,37.254,157.043
C03032=1057.255,347.984,390.293,173.702,37.259,157.044
C03033=1057.263,348.230,390.256,173.706,37.264,157.046
C03034=1057.270,348.477,390.219,173.710,37.270,157.047
C03035=1057.277,348.725,390.182,173.715,37.275,157.048
C03036=1057.284,348.973,390.146,173.719,37.280,157.049
C03037=1057.291,349.219,390.109,173.723,37.284,157.050
C03038=1057.298,349.467,390.072,173.728,37.289,157.052
C03039=1057.304,349.714,390.036,173.731,37.294,157.053
C03040=1057.312,349.961,390.000,173.736,37.299,157.054
C03041=1057.319,350.208,389.962,173.741,37.304,157.055
C03042=1057.326,350.455,389.926,173.745,37.309,157.056
C03043=1057.332,350.703,389.889,173.750,37.314,157.058
C03044=1057.340,350.949,389.852,173.754,37.319,157.059
C03045=1057.347,351.197,389.815,173.759,37.324,157.060
C03046=1057.354,351.444,389.778,173.762,37.329,157.061
C03047=1057.360,351.691,389.741,173.767,37.334,157.062
C03048=1057.368,351.938,389.704,173.771,37.339,157.064
C03049=1057.374,352.186,389.667,173.776,37.344,157.065
C03050=1057.381,352.433,389.630,173.780,37.350,157.066
C03051=1057.388,352.680,389.593,173.785,37.355,157.067
C03052=1057.395,352.927,389.556,173.789,37.360,157.069
C03053=1057.402,353.175,389.519,173.794,37.365,157.070
C03054=1057.409,353.422,389.482,173.797,37.370,157.071
C03055=1057.416,353.668,389.444,173.802,37.375,157.072
C03056=1057.423,353.916,389.408,173.807,37.380,157.073
C03057=1057.430,354.163,389.370,173.811,37.385,157.075
C03058=1057.437,354.410,389.333,173.816,37.390,157.076
C03059=1057.444,354.657,389.295,173.820,37.396,157.077
C03060=1057.451,354.904,389.259,173.825,37.401,157.078
C03061=1057.458,355.152,389.221,173.830,37.406,157.080
C03062=1057.465,355.399,389.184,173.834,37.411,157.081
C03063=1057.472,355.645,389.146,173.838,37.416,157.082
C03064=1057.479,355.892,389.109,173.842,37.422,157.084
C03065=1057.486,356.140,389.072,173.847,37.427,157.085
C03066=1057.493,356.387,389.035,173.852,37.432,157.086
C03067=1057.500,356.634,388.997,173.856,37.438,157.087
C03068=1057.507,356.881,388.960,173.861,37.442,157.089
C03069=1057.514,357.128,388.922,173.866,37.448,157.090
C03070=1057.522,357.375,388.885,173.870,37.453,157.091
C03071=1057.529,357.622,388.847,173.875,37.459,157.092
C03072=1057.536,357.869,388.810,173.880,37.464,157.094
C03073=1057.543,358.116,388.772,173.884,37.469,157.095
C03074=1057.550,358.364,388.734,173.889,37.474,157.096
C03075=1057.556,358.610,388.697,173.894,37.480,157.098
C03076=1057.564,358.857,388.659,173.898,37.485,157.099
C03077=1057.571,359.104,388.622,173.902,37.490,157.100
C03078=1057.578,359.351,388.584,173.907,37.496,157.101
C03079=1057.586,359.610,388.544,173.911,37.501,157.103
C03080=1057.593,359.869,388.504,173.916,37.507,157.104
C03081=1057.600,360.128,388.465,173.922,37.513,157.106
C03082=1057.607,360.387,388.425,173.927,37.518,157.107
C03083=1057.615,360.634,388.388,173.932,37.524,157.108
C03084=1057.622,360.881,388.350,173.937,37.529,157.110
C03085=1057.629,361.128,388.311,173.940,37.534,157.111
C03086=1057.636,361.375,388.274,173.945,37.540,157.112
C03087=1057.644,361.622,388.236,173.950,37.545,157.114
C03088=1057.651,361.869,388.198,173.954,37.551,157.115
C03089=1057.658,362.116,388.159,173.959,37.556,157.116
C03090=1057.665,362.363,388.122,173.964,37.562,157.118
C03091=1057.672,362.610,388.083,173.969,37.567,157.119
C03092=1057.679,362.857,388.045,173.973,37.573,157.120
C03093=1057.686,363.104,388.007,173.978,37.578,157.122
C03094=1057.694,363.351,387.969,173.983,37.584,157.123
C03095=1057.701,363.598,387.930,173.988,37.589,157.124
C03096=1057.708,363.845,387.893,173.993,37.595,157.126
C03097=1057.715,364.092,387.854,173.997,37.600,157.127
C03098=1057.723,364.339,387.816,174.002,37.606,157.128
C03099=1057.729,364.586,387.778,174.007,37.611,157.130
C03100=1057.737,364.833,387.739,174.013,37.618,157.131
C03101=1057.744,365.079,387.701,174.017,37.623,157.133
C03102=1057.751,365.327,387.663,174.022,37.629,157.134
C03103=1057.758,365.573,387.624,174.027,37.635,157.136
C03104=1057.765,365.820,387.586,174.032,37.640,157.137
C03105=1057.772,366.067,387.547,174.037,37.646,157.138
C03106=1057.779,366.314,387.508,174.041,37.651,157.140
C03107=1057.787,366.561,387.470,174.046,37.657,157.141
C03108=1057.793,366.808,387.432,174.051,37.663,157.142
C03109=1057.801,367.055,387.393,174.056,37.669,157.144
C03110=1057.808,367.302,387.354,174.061,37.674,157.145
C03111=1057.815,367.549,387.315,174.066,37.680,157.147
C03112=1057.823,367.796,387.277,174.071,37.686,157.148
C03113=1057.830,368.042,387.238,174.075,37.692,157.150
C03114=1057.837,368.289,387.200,174.080,37.697,157.151
C03115=1057.844,368.536,387.161,174.086,37.703,157.153
C03116=1057.851,368.783,387.122,174.091,37.709,157.154
C03117=1057.859,369.029,387.083,174.096,37.715,157.155
C03118=1057.866,369.276,387.044,174.101,37.720,157.157
C03119=1057.874,369.523,387.006,174.106,37.726,157.158
C03120=1057.881,369.770,386.967,174.111,37.732,157.160
C03121=1057.888,370.017,386.928,174.116,37.738,157.161
C03122=1057.896,370.264,386.889,174.121,37.744,157.163
C03123=1057.903,370.510,386.850,174.125,37.750,157.164
C03124=1057.910,370.757,386.811,174.130,37.755,157.165
C03125=1057.918,371.004,386.772,174.136,37.761,157.167
C03126=1057.925,371.251,386.733,174.141,37.767,157.168
C03127=1057.933,371.498,386.693,174.146,37.773,157.170
C03128=1057.940,371.745,386.655,174.151,37.779,157.171
C03129=1057.947,371.991,386.616,174.156,37.785,157.173
C03130=1057.955,372.238,386.576,174.161,37.791,157.174
C03131=1057.961,372.485,386.538,174.166,37.797,157.176
C03132=1057.969,372.732,386.498,174.172,37.803,157.177
C03133=1057.976,372.979,386.459,174.177,37.809,157.179
C03134=1057.984,373.225,386.420,174.182,37.815,157.180
C03135=1057.992,373.503,386.376,174.187,37.822,157.182
C03136=1058.000,373.780,386.331,174.194,37.828,157.184
C03137=1058.008,374.058,386.287,174.199,37.836,157.186
C03138=1058.017,374.335,386.242,174.205,37.843,157.187
C03139=1058.024,374.582,386.203,174.211,37.849,157.189
C03140=1058.031,374.828,386.163,174.216,37.855,157.190
C03141=1058.038,375.075,386.124,174.221,37.861,157.192
C03142=1058.046,375.322,386.084,174.226,37.867,157.194
C03143=1058.053,375.568,386.045,174.231,37.873,157.195
C03144=1058.061,375.815,386.005,174.237,37.879,157.197
C03145=1058.068,376.062,385.965,174.242,37.886,157.198
C03146=1058.076,376.308,385.925,174.247,37.892,157.200
C03147=1058.083,376.555,385.886,174.252,37.898,157.201
C03148=1058.090,376.802,385.846,174.257,37.904,157.203
C03149=1058.098,377.048,385.806,174.263,37.910,157.204
C03150=1058.105,377.295,385.767,174.268,37.917,157.206
C03151=1058.113,377.542,385.727,174.274,37.923,157.208
C03152=1058.121,377.788,385.687,174.279,37.929,157.209
C03153=1058.128,378.035,385.647,174.285,37.935,157.211
C03154=1058.135,378.282,385.607,174.290,37.942,157.212
C03155=1058.143,378.528,385.567,174.295,37.948,157.214
C03156=1058.150,378.775,385.528,174.300,37.954,157.216
C03157=1058.158,379.022,385.488,174.306,37.961,157.217
C03158=1058.166,379.268,385.448,174.311,37.967,157.219
C03159=1058.173,379.515,385.408,174.317,37.973,157.220
C03160=1058.181,379.761,385.368,174.323,37.980,157.222
C03161=1058.189,380.008,385.328,174.328,37.986,157.224
C03162=1058.196,380.255,385.288,174.333,37.992,157.225
C03163=1058.204,380.502,385.248,174.338,37.999,157.227
C03164=1058.211,380.748,385.207,174.344,38.005,157.229
C03165=1058.218,380.994,385.167,174.350,38.012,157.230
C03166=1058.226,381.241,385.127,174.355,38.018,157.232
C03167=1058.233,381.488,385.086,174.361,38.025,157.234
C03168=1058.241,381.734,385.046,174.366,38.031,157.235
C03169=1058.249,381.980,385.006,174.372,38.038,157.237
C03170=1058.256,382.228,384.965,174.377,38.045,157.239
C03171=1058.264,382.474,384.925,174.383,38.051,157.240
C03172=1058.271,382.720,384.884,174.389,38.058,157.242
C03173=1058.278,382.967,384.844,174.394,38.064,157.244
C03174=1058.286,383.213,384.803,174.399,38.071,157.245
C03175=1058.293,383.460,384.762,174.406,38.078,157.247
C03176=1058.301,383.707,384.722,174.411,38.084,157.249
C03177=1058.309,383.953,384.681,174.416,38.091,157.250
C03178=1058.316,384.199,384.640,174.422,38.098,157.252
C03179=1058.324,384.446,384.600,174.428,38.104,157.254
C03180=1058.332,384.692,384.560,174.434,38.111,157.256
C03181=1058.339,384.938,384.519,174.439,38.118,157.257
C03182=1058.347,385.185,384.478,174.444,38.125,157.259
C03183=1058.354,385.431,384.437,174.451,38.131,157.261
C03184=1058.362,385.678,384.396,174.456,38.138,157.263
C03185=1058.370,385.924,384.356,174.462,38.145,157.264
C03186=1058.377,386.171,384.314,174.468,38.151,157.266
C03187=1058.385,386.417,384.274,174.473,38.158,157.268
C03188=1058.393,386.663,384.233,174.479,38.165,157.270
C03189=1058.401,386.910,384.192,174.485,38.172,157.271
C03190=1058.409,387.157,384.150,174.491,38.178,157.273
C03191=1058.419,387.465,384.100,174.498,38.187,157.275
C03192=1058.428,387.774,384.048,174.505,38.196,157.278
C03193=1058.438,388.083,383.997,174.512,38.205,157.280
C03194=1058.448,388.392,383.945,174.520,38.213,157.282
C03195=1058.455,388.639,383.904,174.526,38.220,157.284
C03196=1058.463,388.885,383.863,174.532,38.227,157.286
C03197=1058.471,389.131,383.823,174.538,38.234,157.288
C03198=1058.479,389.377,383.781,174.544,38.241,157.289
C03199=1058.488,389.624,383.740,174.550,38.248,157.291
C03200=1058.495,389.871,383.698,174.555,38.255,157.293
C03201=1058.503,390.117,383.656,174.562,38.262,157.295
C03202=1058.511,390.363,383.616,174.567,38.269,157.297
C03203=1058.518,390.609,383.574,174.574,38.276,157.299
C03204=1058.526,390.856,383.532,174.579,38.283,157.300
C03205=1058.534,391.102,383.491,174.586,38.291,157.302
C03206=1058.542,391.349,383.450,174.591,38.298,157.304
C03207=1058.549,391.595,383.408,174.598,38.305,157.306
C03208=1058.558,391.841,383.366,174.604,38.312,157.308
C03209=1058.565,392.088,383.325,174.610,38.319,157.310
C03210=1058.573,392.334,383.283,174.616,38.327,157.312
C03211=1058.581,392.579,383.241,174.622,38.333,157.314
C03212=1058.589,392.826,383.200,174.628,38.341,157.316
C03213=1058.597,393.072,383.158,174.635,38.348,157.317
C03214=1058.605,393.319,383.116,174.640,38.355,157.319
C03215=1058.613,393.565,383.074,174.647,38.363,157.321
C03216=1058.620,393.811,383.032,174.652,38.370,157.323
C03217=1058.628,394.058,382.989,174.659,38.378,157.325
C03218=1058.636,394.304,382.947,174.665,38.385,157.327
C03219=1058.644,394.549,382.906,174.671,38.392,157.329
C03220=1058.653,394.796,382.864,174.677,38.400,157.331
C03221=1058.660,395.042,382.822,174.684,38.407,157.333
C03222=1058.668,395.289,382.780,174.690,38.415,157.335
C03223=1058.676,395.535,382.738,174.696,38.422,157.337
C03224=1058.684,395.781,382.695,174.703,38.430,157.339
C03225=1058.692,396.027,382.653,174.708,38.437,157.341
C03226=1058.700,396.274,382.611,174.715,38.444,157.343
C03227=1058.708,396.520,382.569,174.722,38.452,157.345
C03228=1058.716,396.767,382.527,174.728,38.460,157.347
C03229=1058.724,397.012,382.484,174.734,38.467,157.349
C03230=1058.732,397.259,382.442,174.741,38.475,157.351
C03231=1058.740,397.505,382.400,174.747,38.482,157.353
C03232=1058.748,397.751,382.357,174.753,38.490,157.355
C03233=1058.756,397.997,382.315,174.760,38.498,157.357
C03234=1058.764,398.243,382.273,174.766,38.506,157.359
C03235=1058.772,398.489,382.230,174.773,38.513,157.361
C03236=1058.780,398.736,382.187,174.780,38.521,157.363
C03237=1058.788,398.981,382.145,174.785,38.529,157.365
C03238=1058.796,399.228,382.102,174.792,38.537,157.367
C03239=1058.804,399.474,382.059,174.799,38.544,157.369
C03240=1058.812,399.720,382.017,174.806,38.552,157.371
C03241=1058.820,399.967,381.974,174.811,38.560,157.374
C03242=1058.829,400.213,381.931,174.818,38.568,157.376
C03243=1058.837,400.459,381.888,174.825,38.576,157.378
C03244=1058.845,400.706,381.845,174.832,38.584,157.380
C03245=1058.853,400.951,381.802,174.838,38.591,157.382
C03246=1058.861,401.197,381.759,174.845,38.599,157.384
C03247=1058.872,401.524,381.702,174.853,38.610,157.387
C03248=1058.882,401.850,381.646,174.863,38.620,157.390
C03249=1058.894,402.176,381.589,174.871,38.631,157.393
C03250=1058.906,402.502,381.531,174.881,38.641,157.395
C03251=1058.913,402.748,381.488,174.887,38.650,157.398
C03252=1058.921,402.994,381.445,174.893,38.658,157.400
C03253=1058.930,403.240,381.402,174.900,38.666,157.402
C03254=1058.937,403.486,381.358,174.907,38.674,157.404
C03255=1058.946,403.732,381.315,174.914,38.682,157.406
C03256=1058.954,403.979,381.271,174.921,38.690,157.409
C03257=1058.962,404.225,381.228,174.928,38.698,157.411
C03258=1058.971,404.471,381.185,174.935,38.707,157.413
C03259=1058.979,404.716,381.141,174.941,38.715,157.415
C03260=1058.987,404.962,381.098,174.948,38.723,157.418
C03261=1058.995,405.209,381.054,174.955,38.732,157.420
C03262=1059.004,405.455,381.011,174.962,38.740,157.422
C03263=1059.012,405.701,380.967,174.969,38.748,157.424
C03264=1059.021,405.947,380.924,174.976,38.757,157.427
C03265=1059.029,406.193,380.879,174.983,38.765,157.429
C03266=1059.037,406.439,380.836,174.990,38.773,157.431
C03267=1059.045,406.685,380.792,174.997,38.782,157.433
C03268=1059.053,406.931,380.748,175.004,38.790,157.436
C03269=1059.062,407.177,380.704,175.011,38.799,157.438
C03270=1059.070,407.422,380.660,175.018,38.807,157.440
C03271=1059.078,407.669,380.617,175.025,38.816,157.443
C03272=1059.087,407.915,380.572,175.033,38.824,157.445
C03273=1059.095,408.161,380.528,175.040,38.833,157.447
C03274=1059.103,408.407,380.484,175.047,38.842,157.450
C03275=1059.112,408.652,380.441,175.054,38.850,157.452
C03276=1059.121,408.899,380.396,175.061,38.859,157.455
C03277=1059.129,409.145,380.352,175.069,38.867,157.457
C03278=1059.137,409.390,380.308,175.076,38.876,157.459
C03279=1059.146,409.637,380.263,175.083,38.885,157.462
C03280=1059.154,409.882,380.219,175.091,38.894,157.464
C03281=1059.163,410.128,380.175,175.098,38.902,157.466
C03282=1059.172,410.374,380.130,175.105,38.911,157.469
C03283=1059.180,410.620,380.086,175.112,38.920,157.471
C03284=1059.188,410.866,380.041,175.120,38.929,157.474
C03285=1059.197,411.112,379.998,175.128,38.938,157.476
C03286=1059.205,411.358,379.953,175.135,38.946,157.479
C03287=1059.214,411.604,379.909,175.142,38.955,157.481
C03288=1059.223,411.849,379.864,175.149,38.964,157.484
C03289=1059.232,412.095,379.819,175.158,38.973,157.486
C03290=1059.240,412.342,379.775,175.165,38.982,157.489
C03291=1059.248,412.587,379.730,175.172,38.991,157.491
C03292=1059.258,412.833,379.686,175.180,39.000,157.493
C03293=1059.266,413.079,379.641,175.188,39.009,157.496
C03294=1059.275,413.325,379.596,175.195,39.018,157.499
C03295=1059.284,413.571,379.551,175.202,39.027,157.501
C03296=1059.293,413.816,379.507,175.211,39.036,157.504
C03297=1059.302,414.062,379.462,175.218,39.045,157.506
C03298=1059.311,414.308,379.417,175.226,39.054,157.509
C03299=1059.319,414.554,379.372,175.234,39.063,157.511
C03300=1059.328,414.800,379.327,175.241,39.073,157.514
C03301=1059.335,415.045,379.281,175.249,39.082,157.516
C03302=1059.344,415.291,379.236,175.257,39.091,157.519
C03303=1059.357,415.623,379.175,175.267,39.104,157.523
C03304=1059.368,415.954,379.114,175.278,39.116,157.526
C03305=1059.379,416.286,379.053,175.289,39.129,157.530
C03306=1059.392,416.617,378.992,175.299,39.142,157.533
C03307=1059.401,416.863,378.946,175.307,39.151,157.536
C03308=1059.410,417.109,378.901,175.315,39.161,157.539
C03309=1059.418,417.354,378.856,175.324,39.170,157.541
C03310=1059.427,417.600,378.810,175.331,39.180,157.544
C03311=1059.436,417.846,378.765,175.340,39.189,157.547
C03312=1059.445,418.091,378.719,175.347,39.199,157.549
C03313=1059.454,418.337,378.673,175.356,39.209,157.552
C03314=1059.462,418.583,378.627,175.364,39.218,157.555
C03315=1059.471,418.829,378.582,175.372,39.228,157.557
C03316=1059.480,419.074,378.536,175.380,39.238,157.560
C03317=1059.490,419.320,378.490,175.388,39.247,157.563
C03318=1059.499,419.565,378.445,175.397,39.257,157.566
C03319=1059.508,419.811,378.399,175.405,39.267,157.568
C03320=1059.517,420.057,378.353,175.413,39.276,157.571
C03321=1059.526,420.302,378.307,175.421,39.286,157.574
C03322=1059.534,420.548,378.261,175.430,39.296,157.577
C03323=1059.544,420.793,378.215,175.438,39.306,157.580
C03324=1059.552,421.039,378.168,175.447,39.316,157.583
C03325=1059.561,421.284,378.123,175.455,39.326,157.585
C03326=1059.570,421.530,378.076,175.463,39.336,157.588
C03327=1059.580,421.776,378.030,175.472,39.346,157.591
C03328=1059.589,422.021,377.984,175.481,39.356,157.594
C03329=1059.598,422.267,377.937,175.489,39.366,157.597
C03330=1059.607,422.512,377.891,175.498,39.376,157.600
C03331=1059.615,422.757,377.844,175.506,39.387,157.603
C03332=1059.625,423.003,377.797,175.515,39.396,157.605
C03333=1059.634,423.249,377.751,175.523,39.407,157.608
C03334=1059.643,423.494,377.705,175.532,39.417,157.611
C03335=1059.652,423.739,377.658,175.541,39.427,157.614
C03336=1059.662,423.985,377.611,175.550,39.437,157.617
C03337=1059.671,424.231,377.565,175.559,39.448,157.620
C03338=1059.680,424.475,377.518,175.567,39.458,157.623
C03339=1059.690,424.721,377.471,175.576,39.468,157.626
C03340=1059.698,424.967,377.425,175.585,39.479,157.629
C03341=1059.708,425.211,377.378,175.593,39.489,157.632
C03342=1059.717,425.458,377.331,175.602,39.499,157.635
C03343=1059.726,425.703,377.284,175.611,39.510,157.638
C03344=1059.736,425.948,377.237,175.620,39.520,157.641
C03345=1059.745,426.194,377.190,175.629,39.531,157.644
C03346=1059.754,426.439,377.143,175.638,39.542,157.648
C03347=1059.764,426.684,377.095,175.647,39.552,157.651
C03348=1059.773,426.930,377.049,175.656,39.563,157.654
C03349=1059.782,427.176,377.001,175.666,39.574,157.657
C03350=1059.792,427.420,376.954,175.675,39.584,157.660
C03351=1059.802,427.666,376.906,175.684,39.595,157.663
C03352=1059.810,427.911,376.860,175.694,39.606,157.666
C03353=1059.820,428.157,376.812,175.703,39.617,157.669
C03354=1059.830,428.402,376.765,175.712,39.628,157.673
C03355=1059.839,428.647,376.717,175.721,39.638,157.676
C03356=1059.848,428.893,376.669,175.731,39.649,157.679
C03357=1059.858,429.138,376.622,175.740,39.660,157.682
C03358=1059.867,429.382,376.574,175.750,39.671,157.685
C03359=1059.878,429.651,376.522,175.760,39.684,157.689
C03360=1059.888,429.919,376.470,175.771,39.695,157.692
C03361=1059.898,430.188,376.417,175.781,39.707,157.696
C03362=1059.909,430.457,376.365,175.792,39.720,157.700
C03363=1059.919,430.703,376.317,175.801,39.731,157.703
C03364=1059.928,430.947,376.269,175.810,39.742,157.706
C03365=1059.937,431.193,376.221,175.820,39.754,157.710
C03366=1059.947,431.438,376.172,175.830,39.765,157.713
C03367=1059.957,431.683,376.124,175.839,39.776,157.716
C03368=1059.966,431.928,376.076,175.850,39.788,157.720
C03369=1059.976,432.173,376.027,175.859,39.799,157.723
C03370=1059.985,432.419,375.980,175.869,39.810,157.727
C03371=1059.996,432.663,375.932,175.879,39.821,157.730
C03372=1060.005,432.909,375.883,175.888,39.833,157.733
C03373=1060.015,433.154,375.834,175.899,39.845,157.737
C03374=1060.025,433.399,375.786,175.908,39.856,157.740
C03375=1060.034,433.644,375.737,175.919,39.868,157.744
C03376=1060.044,433.889,375.688,175.928,39.880,157.747
C03377=1060.054,434.134,375.640,175.939,39.891,157.751
C03378=1060.064,434.379,375.591,175.949,39.903,157.754
C03379=1060.073,434.624,375.543,175.959,39.914,157.758
C03380=1060.083,434.869,375.494,175.970,39.926,157.761
C03381=1060.093,435.114,375.446,175.979,39.938,157.765
C03382=1060.104,435.359,375.396,175.990,39.949,157.768
C03383=1060.113,435.604,375.348,176.000,39.962,157.772
C03384=1060.123,435.849,375.299,176.011,39.974,157.775
C03385=1060.133,436.093,375.250,176.021,39.985,157.779
C03386=1060.143,436.339,375.201,176.032,39.997,157.783
C03387=1060.154,436.583,375.152,176.042,40.009,157.786
C03388=1060.163,436.828,375.103,176.053,40.021,157.790
C03389=1060.174,437.073,375.054,176.063,40.033,157.794
C03390=1060.184,437.318,375.005,176.073,40.045,157.797
C03391=1060.194,437.563,374.956,176.084,40.057,157.801
C03392=1060.204,437.808,374.906,176.095,40.070,157.805
C03393=1060.214,438.052,374.856,176.106,40.082,157.808
C03394=1060.224,438.297,374.807,176.117,40.094,157.812
C03395=1060.234,438.542,374.757,176.128,40.106,157.816
C03396=1060.244,438.787,374.707,176.138,40.119,157.820
C03397=1060.254,439.031,374.658,176.149,40.131,157.823
C03398=1060.265,439.276,374.609,176.160,40.144,157.827
C03399=1060.274,439.521,374.559,176.171,40.156,157.831
C03400=1060.285,439.766,374.509,176.182,40.169,157.835
C03401=1060.295,440.011,374.459,176.193,40.181,157.839
C03402=1060.305,440.256,374.410,176.204,40.194,157.843
C03403=1060.316,440.500,374.359,176.216,40.207,157.847
C03404=1060.325,440.745,374.309,176.227,40.219,157.850
C03405=1060.336,440.989,374.259,176.238,40.232,157.854
C03406=1060.346,441.234,374.209,176.249,40.245,157.858
C03407=1060.357,441.479,374.159,176.260,40.257,157.862
C03408=1060.367,441.724,374.109,176.271,40.270,157.866
C03409=1060.378,441.968,374.058,176.283,40.283,157.870
C03410=1060.389,442.212,374.008,176.295,40.296,157.874
C03411=1060.399,442.458,373.958,176.306,40.309,157.878
C03412=1060.410,442.702,373.908,176.317,40.322,157.882
C03413=1060.420,442.947,373.857,176.330,40.335,157.886
C03414=1060.430,443.192,373.806,176.341,40.348,157.890
C03415=1060.444,443.526,373.737,176.357,40.366,157.896
C03416=1060.461,443.910,373.658,176.375,40.387,157.903
C03417=1060.478,444.293,373.578,176.394,40.408,157.909
C03418=1060.494,444.676,373.498,176.413,40.428,157.916
C03419=1060.510,445.060,373.418,176.432,40.450,157.922
C03420=1060.522,445.304,373.367,176.443,40.463,157.926
C03421=1060.532,445.548,373.316,176.456,40.477,157.931
C03422=1060.543,445.792,373.264,176.467,40.490,157.935
C03423=1060.554,446.038,373.214,176.480,40.504,157.939
C03424=1060.565,446.282,373.162,176.492,40.518,157.944
C03425=1060.575,446.526,373.111,176.504,40.531,157.948
C03426=1060.586,446.770,373.060,176.517,40.545,157.952
C03427=1060.597,447.015,373.008,176.530,40.558,157.957
C03428=1060.608,447.257,372.957,176.541,40.572,157.961
C03429=1060.620,447.501,372.906,176.554,40.586,157.965
C03430=1060.632,447.745,372.857,176.567,40.599,157.970
C03431=1060.646,447.990,372.807,176.579,40.612,157.974
C03432=1060.661,448.234,372.758,176.592,40.625,157.978
C03433=1060.676,448.477,372.710,176.605,40.638,157.982
C03434=1060.692,448.723,372.662,176.618,40.650,157.986
C03435=1060.709,448.968,372.615,176.631,40.662,157.990
C03436=1060.728,449.212,372.568,176.644,40.674,157.994
C03437=1060.746,449.457,372.523,176.657,40.685,157.998
C03438=1060.765,449.702,372.477,176.671,40.697,158.002
C03439=1060.787,449.948,372.433,176.684,40.708,158.005
C03440=1060.455,449.960,372.156,176.679,40.822,158.037
C03441=1060.434,449.714,372.201,176.665,40.811,158.033
C03442=1060.414,449.468,372.245,176.651,40.800,158.029
C03443=1060.395,449.223,372.291,176.638,40.788,158.025
C03444=1060.377,448.978,372.337,176.625,40.776,158.021
C03445=1060.360,448.733,372.385,176.612,40.764,158.017
C03446=1060.343,448.489,372.432,176.599,40.752,158.013
C03447=1060.328,448.244,372.481,176.586,40.740,158.009
C03448=1060.313,448.000,372.529,176.573,40.727,158.005
C03449=1060.299,447.756,372.578,176.560,40.714,158.001
C03450=1060.287,447.512,372.629,176.548,40.700,157.997
C03451=1060.275,447.269,372.679,176.535,40.687,157.992
C03452=1060.264,447.026,372.731,176.522,40.674,157.988
C03453=1060.252,446.782,372.782,176.510,40.660,157.984
C03454=1060.242,446.537,372.833,176.498,40.646,157.979
C03455=1060.231,446.293,372.885,176.485,40.633,157.975
C03456=1060.219,446.048,372.936,176.473,40.619,157.971
C03457=1060.209,445.803,372.987,176.461,40.605,157.966
C03458=1060.199,445.559,373.039,176.448,40.592,157.962
C03459=1060.187,445.316,373.090,176.436,40.578,157.958
C03460=1060.177,445.071,373.140,176.424,40.565,157.953
C03461=1060.161,444.707,373.217,176.406,40.545,157.947
C03462=1060.145,444.343,373.293,176.388,40.526,157.941
C03463=1060.129,443.978,373.368,176.371,40.506,157.935
C03464=1060.113,443.615,373.444,176.353,40.486,157.929
C03465=1060.103,443.370,373.495,176.340,40.473,157.924
C03466=1060.092,443.125,373.545,176.329,40.460,157.920
C03467=1060.082,442.881,373.596,176.318,40.447,157.916
C03468=1060.071,442.636,373.646,176.305,40.434,157.912
C03469=1060.061,442.391,373.697,176.294,40.421,157.908
C03470=1060.050,442.147,373.747,176.283,40.408,157.904
C03471=1060.040,441.902,373.797,176.270,40.395,157.900
C03472=1060.029,441.658,373.848,176.259,40.382,157.896
C03473=1060.019,441.413,373.898,176.248,40.370,157.892
C03474=1060.008,441.168,373.948,176.237,40.357,157.888
C03475=1059.998,440.924,373.999,176.226,40.344,157.884
C03476=1059.988,440.679,374.048,176.213,40.332,157.880
C03477=1059.977,440.435,374.099,176.202,40.319,157.876
C03478=1059.967,440.189,374.149,176.191,40.307,157.872
C03479=1059.957,439.945,374.198,176.180,40.294,157.869
C03480=1059.947,439.700,374.249,176.169,40.281,157.865
C03481=1059.936,439.455,374.299,176.158,40.269,157.861
C03482=1059.926,439.211,374.348,176.147,40.257,157.857
C03483=1059.915,438.966,374.398,176.136,40.244,157.853
C03484=1059.906,438.721,374.447,176.125,40.232,157.849
C03485=1059.895,438.476,374.497,176.114,40.219,157.846
C03486=1059.885,438.232,374.546,176.103,40.207,157.842
C03487=1059.875,437.986,374.596,176.092,40.195,157.838
C03488=1059.865,437.742,374.646,176.081,40.183,157.834
C03489=1059.855,437.497,374.695,176.071,40.171,157.831
C03490=1059.845,437.252,374.744,176.060,40.158,157.827
C03491=1059.834,437.007,374.793,176.050,40.146,157.823
C03492=1059.825,436.762,374.843,176.039,40.134,157.820
C03493=1059.811,436.439,374.907,176.025,40.119,157.815
C03494=1059.798,436.114,374.972,176.011,40.103,157.810
C03495=1059.784,435.791,375.037,175.997,40.087,157.805
C03496=1059.771,435.467,375.102,175.983,40.072,157.801
C03497=1059.761,435.222,375.151,175.973,40.060,157.797
C03498=1059.752,434.977,375.199,175.963,40.048,157.793
C03499=1059.742,434.732,375.249,175.952,40.037,157.790
C03500=1059.732,434.487,375.298,175.942,40.024,157.786
C03501=1059.722,434.242,375.346,175.932,40.013,157.783
C03502=1059.712,433.997,375.395,175.921,40.001,157.779
C03503=1059.703,433.752,375.443,175.912,39.990,157.776
C03504=1059.693,433.507,375.492,175.901,39.978,157.772
C03505=1059.683,433.262,375.540,175.891,39.967,157.769
C03506=1059.673,433.017,375.589,175.881,39.956,157.765
C03507=1059.664,432.772,375.638,175.871,39.944,157.762
C03508=1059.654,432.527,375.686,175.861,39.932,157.758
C03509=1059.644,432.282,375.735,175.852,39.921,157.755
C03510=1059.635,432.037,375.782,175.841,39.910,157.752
C03511=1059.625,431.792,375.831,175.832,39.898,157.748
C03512=1059.615,431.547,375.879,175.821,39.887,157.745
C03513=1059.606,431.301,375.927,175.812,39.876,157.742
C03514=1059.596,431.056,375.976,175.802,39.864,157.738
C03515=1059.586,430.811,376.024,175.792,39.853,157.735
C03516=1059.577,430.566,376.071,175.783,39.842,157.732
C03517=1059.565,430.291,376.125,175.772,39.830,157.728
C03518=1059.555,430.015,376.179,175.761,39.817,157.724
C03519=1059.544,429.740,376.233,175.751,39.805,157.721
C03520=1059.533,429.464,376.287,175.740,39.792,157.717
C03521=1059.524,429.219,376.334,175.730,39.782,157.714
C03522=1059.514,428.974,376.382,175.720,39.771,157.710
C03523=1059.505,428.728,376.430,175.711,39.760,157.707
C03524=1059.495,428.483,376.477,175.702,39.749,157.704
C03525=1059.486,428.238,376.525,175.693,39.738,157.701
C03526=1059.476,427.992,376.572,175.683,39.728,157.698
C03527=1059.467,427.748,376.619,175.674,39.717,157.695
C03528=1059.457,427.502,376.667,175.664,39.706,157.691
C03529=1059.448,427.256,376.715,175.655,39.695,157.688
C03530=1059.438,427.012,376.762,175.646,39.685,157.685
C03531=1059.429,426.766,376.809,175.637,39.674,157.682
C03532=1059.420,426.521,376.856,175.628,39.663,157.679
C03533=1059.410,426.275,376.903,175.619,39.653,157.676
C03534=1059.402,426.030,376.950,175.610,39.642,157.673
C03535=1059.391,425.785,376.997,175.601,39.632,157.670
C03536=1059.383,425.539,377.044,175.592,39.621,157.667
C03537=1059.373,425.294,377.091,175.583,39.611,157.664
C03538=1059.364,425.048,377.138,175.574,39.600,157.660
C03539=1059.354,424.803,377.185,175.565,39.590,157.658
C03540=1059.345,424.558,377.232,175.556,39.580,157.655
C03541=1059.336,424.312,377.279,175.547,39.570,157.652
C03542=1059.327,424.066,377.325,175.538,39.559,157.649
C03543=1059.317,423.822,377.372,175.529,39.549,157.646
C03544=1059.308,423.576,377.419,175.520,39.539,157.643
C03545=1059.299,423.330,377.465,175.511,39.529,157.640
C03546=1059.290,423.085,377.511,175.503,39.518,157.637
C03547=1059.281,422.839,377.559,175.494,39.508,157.634
C03548=1059.271,422.594,377.605,175.486,39.498,157.631
C03549=1059.263,422.348,377.651,175.477,39.488,157.628
C03550=1059.253,422.103,377.698,175.468,39.478,157.625
C03551=1059.244,421.858,377.744,175.459,39.468,157.622
C03552=1059.235,421.611,377.791,175.451,39.458,157.619
C03553=1059.226,421.366,377.837,175.443,39.448,157.616
C03554=1059.217,421.121,377.884,175.434,39.438,157.614
C03555=1059.208,420.875,377.929,175.425,39.429,157.611
C03556=1059.199,420.630,377.975,175.418,39.419,157.608
C03557=1059.190,420.384,378.022,175.409,39.408,157.605
C03558=1059.181,420.138,378.067,175.400,39.399,157.602
C03559=1059.172,419.893,378.113,175.393,39.389,157.599
C03560=1059.163,419.647,378.159,175.384,39.379,157.597
C03561=1059.154,419.402,378.205,175.375,39.370,157.594
C03562=1059.146,419.156,378.251,175.368,39.360,157.591
C03563=1059.136,418.911,378.297,175.359,39.350,157.588
C03564=1059.127,418.665,378.343,175.350,39.341,157.586
C03565=1059.118,418.419,378.388,175.343,39.331,157.583
C03566=1059.109,418.174,378.434,175.334,39.322,157.580
C03567=1059.100,417.928,378.480,175.327,39.312,157.578
C03568=1059.091,417.682,378.525,175.318,39.303,157.575
C03569=1059.082,417.436,378.570,175.309,39.293,157.572
C03570=1059.073,417.191,378.616,175.302,39.283,157.569
C03571=1059.065,416.945,378.663,175.293,39.274,157.567
C03572=1059.056,416.699,378.708,175.286,39.265,157.564
C03573=1059.044,416.366,378.769,175.275,39.252,157.561
C03574=1059.032,416.032,378.831,175.264,39.239,157.557
C03575=1059.020,415.699,378.892,175.254,39.226,157.553
C03576=1059.008,415.365,378.953,175.242,39.214,157.550
C03577=1058.999,415.119,378.999,175.235,39.205,157.547
C03578=1058.991,414.874,379.044,175.227,39.195,157.545
C03579=1058.982,414.628,379.089,175.219,39.186,157.542
C03580=1058.973,414.382,379.134,175.212,39.177,157.539
C03581=1058.965,414.137,379.179,175.203,39.168,157.537
C03582=1058.956,413.891,379.224,175.196,39.159,157.534
C03583=1058.947,413.645,379.269,175.188,39.149,157.532
C03584=1058.939,413.399,379.314,175.180,39.141,157.529
C03585=1058.930,413.153,379.359,175.173,39.131,157.527
C03586=1058.920,412.907,379.404,175.165,39.122,157.524
C03587=1058.912,412.662,379.448,175.157,39.114,157.522
C03588=1058.903,412.416,379.493,175.150,39.105,157.519
C03589=1058.894,412.170,379.537,175.142,39.096,157.517
C03590=1058.886,411.924,379.582,175.135,39.087,157.514
C03591=1058.878,411.678,379.626,175.127,39.078,157.512
C03592=1058.869,411.432,379.672,175.120,39.069,157.509
C03593=1058.860,411.187,379.715,175.112,39.060,157.507
C03594=1058.851,410.941,379.760,175.105,39.051,157.504
C03595=1058.843,410.695,379.804,175.097,39.043,157.502
C03596=1058.834,410.449,379.848,175.089,39.034,157.499
C03597=1058.826,410.203,379.893,175.082,39.025,157.497
C03598=1058.817,409.956,379.938,175.075,39.016,157.495
C03599=1058.809,409.711,379.982,175.068,39.007,157.492
C03600=1058.800,409.465,380.026,175.061,38.999,157.490
C03601=1058.791,409.219,380.070,175.053,38.990,157.487
C03602=1058.783,408.973,380.115,175.045,38.982,157.485
C03603=1058.775,408.728,380.158,175.038,38.973,157.483
C03604=1058.766,408.481,380.203,175.031,38.965,157.480
C03605=1058.758,408.235,380.247,175.024,38.956,157.478
C03606=1058.749,407.990,380.291,175.017,38.947,157.476
C03607=1058.741,407.744,380.335,175.010,38.939,157.473
C03608=1058.732,407.498,380.379,175.002,38.930,157.471
C03609=1058.724,407.252,380.423,174.995,38.922,157.469
C03610=1058.716,407.005,380.467,174.988,38.914,157.466
C03611=1058.707,406.760,380.511,174.981,38.905,157.464
C03612=1058.699,406.514,380.555,174.974,38.897,157.462
C03613=1058.691,406.268,380.599,174.967,38.888,157.459
C03614=1058.682,406.022,380.643,174.960,38.880,157.457
C03615=1058.674,405.775,380.686,174.953,38.872,157.455
C03616=1058.665,405.530,380.730,174.946,38.863,157.453
C03617=1058.658,405.284,380.774,174.939,38.855,157.450
C03618=1058.649,405.038,380.817,174.932,38.847,157.448
C03619=1058.641,404.792,380.861,174.925,38.838,157.446
C03620=1058.633,404.546,380.904,174.918,38.830,157.443
C03621=1058.625,404.299,380.948,174.911,38.822,157.441
C03622=1058.616,404.053,380.991,174.904,38.814,157.439
C03623=1058.608,403.808,381.034,174.898,38.806,157.437
C03624=1058.600,403.562,381.078,174.891,38.797,157.435
C03625=1058.591,403.315,381.121,174.884,38.789,157.432
C03626=1058.583,403.069,381.165,174.877,38.781,157.430
C03627=1058.575,402.823,381.208,174.870,38.773,157.428
C03628=1058.566,402.577,381.251,174.863,38.765,157.426
C03629=1058.556,402.249,381.309,174.854,38.754,157.423
C03630=1058.545,401.921,381.366,174.845,38.744,157.420
C03631=1058.534,401.593,381.423,174.836,38.733,157.417
C03632=1058.523,401.265,381.481,174.828,38.723,157.414
C03633=1058.515,401.019,381.523,174.821,38.715,157.412
C03634=1058.506,400.773,381.566,174.814,38.707,157.410
C03635=1058.498,400.527,381.609,174.807,38.699,157.408
C03636=1058.489,400.280,381.652,174.800,38.691,157.406
C03637=1058.483,400.034,381.695,174.794,38.684,157.404
C03638=1058.474,399.788,381.738,174.787,38.676,157.402
C03639=1058.466,399.542,381.781,174.781,38.668,157.400
C03640=1058.457,399.295,381.823,174.774,38.660,157.398
